	IF Execute
	THEN
		Error												:=	FALSE;
		ErrorId												:= 0;
		CfgReconfigGroup.bExecute 							:= TRUE;
	ELSIF NOT CfgReconfigGroup.bBusy    					
	THEN                                					
		Error												:=	FALSE;
		ErrorId												:= 0;
		CfgReconfigGroup.bExecute 							:= FALSE;

	END_IF

	CfgReconfigGroup(
		bExecute	:= ,
		nGroupId	:= rNCIRef.NciToPlc.GrpId,
		tTimeOut	:= ,
		bBusy		=> busy,
		bErr		=> ,
		nErrId		=> );

	Done													:= NOT CfgReconfigGroup.bBusy
																AND NOT CfgReconfigGroup.bErr
																AND CfgReconfigGroup.bExecute;
                                        					
	IF NOT Busy
	THEN
		IF CfgReconfigGroup.bExecute
		THEN
			Error											:=	CfgReconfigGroup.bErr;
			ErrorId											:= CfgReconfigGroup.nErrId;
			ErrorText										:= SEL(Error , '' ,  CONCAT('Error CfgReconfigGroup id: ',  UDINT_TO_STRING(Errorid)));
		END_IF                      						
		IF NOT Execute              						
		THEN                        						
			MemFnc											:= -1 ;
			CfgReconfigGroup(bExecute := FALSE,);
		END_IF
	END_IF
	
	Reconfig												:= Busy;
END_METHOD

METHOD PUBLIC reconfigAxis : BOOL //Return value = TRUE if busy
//required parameter
//rNCIRef
//AxisId
VAR_INPUT
	Execute													:	BOOL;
	AxisId													:	UDINT; //Axis ID which should be released from group - if 0 then ID of input parameters is used based on parameter AxisIndex
END_VAR
	MemFnc													:= FNC_ADD_AXIS;
	THIS^.Execute											:= Execute;
	
IF NOT __ISVALIDREF(rNCIRef) THEN
	Busy													:= NOT Error;
	Error													:= TRUE;
	ErrorId													:= E_AdsErr.DEVICE_INVALIDPARM;
	Done													:= FALSE;
	ErrorText												:= 'Reference to rNCIRef invalid (0)';
	MemFnc													:= SEL(Execute , -1 ,MemFnc);
	RETURN;
END_IF

	IF Execute
	THEN
		Error												:=	FALSE;
		ErrorId												:= 0;
		CfgReconfigAxis.bExecute 							:= TRUE;
	ELSIF NOT CfgReconfigAxis.bBusy     					
	THEN                                					
		Error												:=	FALSE;
		ErrorId												:= 0;
		CfgReconfigAxis.bExecute 							:= FALSE;

	END_IF

	IF AxisId > 0
	THEN
		CfgReconfigAxis.nAxisId								:= AxisId;
	ELSE
		CASE AxisIndex OF
		1:	CfgReconfigAxis.nAxisId 						:= XAxisId ;
		2:	CfgReconfigAxis.nAxisId 						:= YAxisId ;
		3:	CfgReconfigAxis.nAxisId 						:= ZAxisId ;
		4:	CfgReconfigAxis.nAxisId 						:= Q1AxisId ;
		5:	CfgReconfigAxis.nAxisId 						:= Q2AxisId ;
		6:	CfgReconfigAxis.nAxisId 						:= Q3AxisId ;
		7:	CfgReconfigAxis.nAxisId 						:= Q4AxisId ;
		8:	CfgReconfigAxis.nAxisId 						:= Q5AxisId ;
		ELSE
			CfgReconfigAxis.nAxisId 						:= 0;
		END_CASE
	END_IF

	CfgReconfigAxis(
		bExecute	:= ,
		nAxisId		:= ,
		tTimeOut	:= ,
		bBusy		=> busy,
		bErr		=> ,
		nErrId		=> );

	Done													:= NOT CfgReconfigAxis.bBusy
																AND NOT CfgReconfigAxis.bErr
																AND CfgReconfigAxis.bExecute;
                                        					
	IF NOT Busy
	THEN
		IF CfgReconfigAxis.bExecute
		THEN
			Error											:=	CfgReconfigAxis.bErr;
			ErrorId											:= CfgReconfigAxis.nErrId;
			ErrorText										:= SEL(Error , '' ,  CONCAT('Error CfgReconfigAxis id: ',  UDINT_TO_STRING(Errorid)));
		END_IF
		IF NOT Execute
		THEN
			MemFnc											:= -1 ;
			CfgReconfigAxis(bExecute := FALSE);
		END_IF
	END_IF
	
	ReconfigAxis											:= Busy;
END_METHOD

END_FUNCTION_BLOCK

// POUs/Motion/TF5100-NCI/01_Main/NciItp
//Nci Interpolation group control - load,start,stop Nci programs as well start interpolated moves via Plc table (Tc2_PlcInterpolation library)
//based on Tc2_NCI, TcNcCfg.lib, Tc2_PlcInterpolation librarys
FUNCTION_BLOCK NciItp  EXTENDS FbBase
VAR_OUTPUT CONSTANT
	FNC_RESET												:	INT := 0; //Reset Nci group
	FNC_LOAD												:	INT := 1; //Load Nci program as txt/nc file
	FNC_START												:	INT := 2; //Start loaded Nci program
	FNC_STOP												:	INT := 3; //Stop loaded Nci programm
	FNC_FEED_TBL											:	INT := 4; //Feed table group - provided by Tc2_PlcInterpolation library
END_VAR                     								
VAR_INPUT                   								
	Fnc														:	INT (FNC_RESET..FNC_FEED_TBL):= FNC_RESET;
	Prg														:	T_MaxString := '';	//Program
	rTable													:	REFERENCE TO ST_NciFeedGroupTable := 0; //-> NciItpTableEntry
	rNCIRef													:	REFERENCE TO NCI_REF := 0;
	StartPrgAfterLoading									:	BOOL := FALSE; //Return value TRUE = Start Program direct after loading 
	LogFeederEntries										:	BOOL := FALSE; //Return value TRUE = Log tabel entries by Fnc FeedTbl
	WaitForChnDoneByEndOfTbl								:	BOOL := FALSE; //Fnc FeedTabl - TRUE = FB is busy as long as the prg is running if table contains entry "ST_NciEndOfTables"
END_VAR                     								
VAR_IN_OUT                  								
END_VAR                     								
VAR_OUTPUT                  								
	ErrorText												:	STRING(40);
END_VAR
VAR
(* cache **************************************************************************)
	MemFnc													:	INT := -1;
	MemResetAfterStop										:	BOOL;
                            								
(* timer *)                 								
                            	
(* trigger *)               	

(* MC-Function-block intances ******************************************************)
	ItpLoadProgEx											:	ItpLoadProgEx;
	ItpStartStopEx											:	ItpStartStopEx;
	NciFeedTable											:	FB_NciFeedTable;
	ItpResetEx2												:	ItpResetEx2 := (tTimeOut	:= DEFAULT_ADS_TIMEOUT);

END_VAR

	(* NCI Program control																*)
	(************************************************************************************)

(* Execute ***************************************************************************************)
	rtExecute(CLK := Execute );
	IF rtExecute.Q
		AND MemFnc < 0
	THEN
		MemFnc 												:= Fnc;
		Busy												:= TRUE;
		Done												:= FALSE;
		Error												:= FALSE;
		ErrorID												:= 0;
		ErrorText											:= '';
	END_IF

(* Call Method ***********************************************************************************)
	CASE MemFnc OF
	FNC_RESET							:
		Reset(Execute:= Execute);
	FNC_LOAD							:
		LoadPrg(Execute:= Execute, Prg:= Prg);
	FNC_START							:
		StartPrg(Execute:= Execute);
	FNC_STOP							:
		StopPrg(Execute:= Execute);
	FNC_FEED_TBL						:
		FeedTbl(Execute:= Execute );
	-1:
		IF NOT Execute
		THEN
			Busy											:= FALSE;
			Done											:= FALSE;
			Error											:= FALSE;
			ErrorID											:= 0;
			ErrorText										:= '';
		END_IF                              				
	ELSE                                    				
		Busy												:= FALSE;
		Done												:= FALSE;
		Error												:= Execute;
		ErrorID												:= E_AdsErr.DEVICE_INVALIDPARM;
		ErrorText											:= CONCAT('invalid parameter value(s) Fnc no: ' , INT_TO_STRING(MemFnc));
	END_CASE


(**************************************************************************************************)

METHOD PUBLIC feedTbl : BOOL //Return value = TRUE if busy
//required parameter
//rNCIRef
//rTable
VAR_INPUT
	Execute													:	BOOL := FALSE;
END_VAR
	MemFnc													:= FNC_FEED_TBL;
	THIS^.Execute											:= Execute;
	
IF NOT __ISVALIDREF(rNCIRef) 
THEN
	Busy													:= NOT Error;
	Error													:= TRUE;
	ErrorId													:= E_AdsErr.DEVICE_INVALIDPARM;
	Done													:= FALSE;
	ErrorText												:= 'Reference rNCIRef invalid (0)';
	MemFnc													:= SEL(Execute , -1 ,MemFnc); 
	RETURN;
ELSIF NOT __ISVALIDREF(rTable) 
THEN
	Busy													:= NOT Error;
	Error													:= TRUE;
	ErrorId													:= E_AdsErr.DEVICE_INVALIDPARM;
	Done													:= FALSE;
	ErrorText												:= 'Reference rTable invalid (0)';
	MemFnc													:= SEL(Execute , -1 ,MemFnc);
	RETURN;
END_IF

	IF Execute
	THEN
		Error												:=	FALSE;
		ErrorId												:= 0;
		NciFeedTable.bExecute 								:= TRUE;
	ELSIF NOT NciFeedTable.bFeedBusy
		AND(
		NOT NciFeedTable.bExecChannelDoneCheck
		OR NciFeedTable.bChannelDone)
	THEN
		Error												:=	FALSE;
		ErrorId												:= 0;
		NciFeedTable.bExecute 								:= FALSE;
	END_IF

	NciFeedTable(
		bExecute			:= ,
		bReset				:= FALSE,
		bLogFeederEntries	:= LogFeederEntries,
		stFeedGroupTable	:= rTable,
		stNciToPlc			:= rNCIRef.NciToPlc,
		bFeedingDone		=> 	,
		bChannelDone		=> ,
		bFeedBusy			=> ,
		bResetBusy			=> ,
		bError				=> ,
		nErrorId			=> );

	IF WaitForChnDoneByEndOfTbl
	THEN
		Busy 												:= NciFeedTable.bFeedBusy
																OR
																NciFeedTable.bFeedingDone
																AND NciFeedTable.bExecChannelDoneCheck
																AND NOT NciFeedTable.bChannelDone;
                            								
		Done												:= NciFeedTable.bChannelDone
																OR
																NciFeedTable.bFeedingDone
																AND NOT NciFeedTable.bExecChannelDoneCheck;
                            								
	ELSE                    								
		Busy												:= NciFeedTable.bFeedBusy;
		Done												:= NciFeedTable.bFeedingDone;
	END_IF

	IF NOT Busy
	THEN
		IF NciFeedTable.bExecute
		THEN
			Error											:=	NciFeedTable.bError;
			ErrorId											:= NciFeedTable.nErrorId;
			ErrorText										:= SEL(Error , '' ,  CONCAT('Error NciFeedTable id: ',  UDINT_TO_STRING(Errorid)));
		END_IF                          					
		IF NOT Execute                  					
		THEN                            					
			MemFnc											:= -1 ;
			NciFeedTable(bExecute 							:= FALSE, stNciToPlc:= rNCIRef.NciToPlc, stFeedGroupTable:= rTable  );
		END_IF                          	
	END_IF                              	
                                        	
	FeedTbl													:= Busy;
END_METHOD

METHOD PUBLIC loadPrg : BOOL //Return value = TRUE if busy
//required parameter
//rNCIRef
VAR_INPUT
	Execute													:	BOOL;
	Prg														:	T_MaxString := ''; //if Prg = '' then INPUT THIS^.Prg used
END_VAR
	MemFnc													:= FNC_LOAD;
	THIS^.Execute											:= Execute;
	
IF NOT __ISVALIDREF(rNCIRef) THEN
	Busy													:= NOT Error;
	Error													:= TRUE;
	ErrorId													:= E_AdsErr.DEVICE_INVALIDPARM;
	Done													:= FALSE;
	ErrorText												:= 'Reference rNCIRef invalid (0)';
	MemFnc													:= SEL(Execute , -1 ,MemFnc);
	RETURN;
END_IF
	
	IF Execute AND NOT ItpLoadProgEx.bExecute
	THEN
		IF LEN(Prg) > 0
		THEN
			ItpLoadProgEx.sPrg								:= Prg;
		ELSE                    							
			ItpLoadProgEx.sPrg								:= THIS^.Prg;	
		END_IF
	END_IF	
	
	IF Execute
	THEN
		Error												:=	FALSE;
		ErrorId												:= 0;
		ItpLoadProgEx.bExecute 								:= TRUE;
	ELSIF NOT ItpLoadProgEx.bBusy       					
		AND(                            					
		NOT ItpStartStopEx.bBusy        					
		OR NOT StartPrgAfterLoading)    					
	THEN                                					
		Error												:=	FALSE;
		ErrorId												:= 0;
		ItpLoadProgEx.bExecute 								:= FALSE;
		IF StartPrgAfterLoading             				
		THEN                                				
			ItpStartStopEx.bStart 							:= FALSE;
		END_IF
	END_IF
	
	ItpLoadProgEx(
		bExecute	:= ,
		sPrg		:= ,
		nLength		:= INT_TO_UDINT(LEN(Prg)),
		tTimeOut	:= ,
		sNciToPlc	:= rNCIRef.NciToPlc,
		bBusy		=> ,
		bErr		=> ,
		nErrId		=> );

	IF StartPrgAfterLoading
		OR ItpStartStopEx.bBusy
	THEN
		ItpStartStopEx(
			bStart		:= ItpLoadProgEx.bExecute
							AND NOT ItpLoadProgEx.bErr
							AND NOT ItpLoadProgEx.bBusy,
			bStop		:= FALSE,
			tTimeOut	:=  ,
			sNciToPlc	:= rNCIRef.NciToPlc,
			bBusy		=> ,
			bErr		=> ,
			nErrId		=> );
	END_IF


	Busy													:= ItpStartStopEx.bBusy OR ItpLoadProgEx.bBusy;
                                        					
	IF StartPrgAfterLoading             					
	THEN                                					
		Done												:= NOT Busy
																AND NOT ItpStartStopEx.bErr
																AND ItpStartStopEx.bStart;
	ELSE                                	    		
		Done												:= NOT Busy
																AND NOT ItpLoadProgEx.bErr
																AND ItpLoadProgEx.bExecute;
	END_IF                                      		
                                                	
	IF NOT Busy                                 	
	THEN
		IF ItpLoadProgEx.bExecute
			AND NOT StartPrgAfterLoading
		THEN
			Error											:=	ItpLoadProgEx.bErr;
			ErrorId											:= ItpLoadProgEx.nErrId;
			ErrorText										:= SEL(Error , '' ,  CONCAT('Error ItpLoadProgEx id: ',  UDINT_TO_STRING(Errorid)));
		ELSIF ItpStartStopEx.bStart 						
		THEN                        						
			Error												:=	ItpStartStopEx.bErr;
			ErrorId											:= ItpStartStopEx.nErrId;
			ErrorText										:= SEL(Error , '' ,  CONCAT('Error ItpStartStopEx id: ',  UDINT_TO_STRING(Errorid)));
		END_IF                          					
                                        					
		IF NOT Execute                  	
		THEN                            	
			MemFnc											:= -1 ;
			ItpLoadProgEx(bExecute := FALSE, sNciToPlc:= rNCIRef.NciToPlc);
			IF StartPrgAfterLoading
			THEN
				ItpStartStopEx(bStart := FALSE, sNciToPlc:= rNCIRef.NciToPlc);
			END_IF
		END_IF
	END_IF
	
	LoadPrg													:= Busy;
END_METHOD

METHOD PUBLIC reset : BOOL //Return value = TRUE if busy
//required parameter
//rNCIRef
//rTable
VAR_INPUT	
	Execute													:	BOOL := FALSE;
END_VAR
	MemFnc													:= FNC_RESET;
	THIS^.Execute											:= Execute;
	
IF NOT __ISVALIDREF(rNCIRef) 
THEN
	Busy													:= NOT Error;
	Error													:= TRUE;
	ErrorId													:= E_AdsErr.DEVICE_INVALIDPARM;
	Done													:= FALSE;
	ErrorText												:= 'Reference rNCIRef invalid (0)';
	MemFnc													:= SEL(Execute , -1 ,MemFnc);
	RETURN;
ELSIF NOT __ISVALIDREF(rTable) AND FALSE 
THEN
	Busy													:= NOT Error;
	Error													:= TRUE;
	ErrorId													:= E_AdsErr.DEVICE_INVALIDPARM;
	Done													:= FALSE;
	ErrorText												:= 'Reference rTable invalid (0)';
	MemFnc													:= SEL(Execute , -1 ,MemFnc);
	RETURN;
END_IF

IF Execute
THEN
	Error													:=	FALSE;
	ErrorId													:= 0;
	NciFeedTable.bReset 									:= __ISVALIDREF(rTable);
	ItpResetEx2.bExecute									:= NOT __ISVALIDREF(rTable);
ELSIF NOT NciFeedTable.bFeedBusy                        	
AND NOT ItpResetEx2.bBusy                               	
THEN                                                    	
	Error													:=	FALSE;
	ErrorId													:= 0;
	NciFeedTable.bReset 									:= FALSE;
	ItpResetEx2.bExecute									:= FALSE; 
END_IF

IF	NOT __ISVALIDREF(rTable)
THEN
	ItpResetEx2(
		bExecute	:= ,
		tTimeOut	:= ,
		sNciToPlc	:= rNCIRef.NciToPlc,
		bBusy		=> Busy,
		bErr		=> ,
		nErrId		=> );
ELSE
	NciFeedTable(
		bExecute			:= FALSE,
		bReset				:= ,
		bLogFeederEntries	:= ,
		stFeedGroupTable	:= rTable,
		stNciToPlc			:= rNCIRef.NciToPlc,
		bFeedingDone		=> ,
		bChannelDone		=> ,
		bFeedBusy			=> ,
		bResetBusy			=> busy,
		bError				=> ,
		nErrorId			=> );
END_IF
Done														:= NOT NciFeedTable.bResetBusy AND NOT ItpResetEx2.bBusy
															 	AND NOT NciFeedTable.bError AND NOT ItpResetEx2.bErr
															 	AND(NciFeedTable.bReset OR ItpResetEx2.bExecute);
                                                      	     
IF NOT Busy                                           	     
THEN                                                  	     
	IF NciFeedTable.bReset                            	     
	THEN                                              	     
		Error												 :=	NciFeedTable.bError;
		ErrorId												 := NciFeedTable.nErrorId;
		ErrorText											 := SEL(Error , '' ,  CONCAT('Error NciFeedTable id: ',  UDINT_TO_STRING(Errorid)));
	ELSIF ItpResetEx2.bExecute      						 
	THEN                            						 
		Error												 :=	ItpResetEx2.bErr;
		ErrorId												 := ItpResetEx2.nErrId;
		ErrorText											 := SEL(Error , '' ,  CONCAT('Error ItpResetEx2 id: ',  UDINT_TO_STRING(Errorid)));		
	END_IF                                            	     
	IF NOT Execute                                    	     
	THEN                                                	
		MemFnc												:= -1 ;
		IF	NOT __ISVALIDREF(rTable)                    	
		THEN                                            	
			ItpResetEx2(bExecute							:= FALSE,sNciToPlc:= rNCIRef.NciToPlc);
		ELSE                                            	
			NciFeedTable(bReset 							:= FALSE, stNciToPlc:= rNCIRef.NciToPlc,stFeedGroupTable:= rTable );
		END_IF                                          	
	END_IF                                              	
END_IF                                                  	
                                                        	
Reset														:= Busy;
END_METHOD

METHOD PUBLIC startPrg : BOOL //Return value = TRUE if busy
//required parameter
//rNCIRef
VAR_INPUT
	Execute													:	BOOL;
END_VAR
	MemFnc													:= FNC_START;
	THIS^.Execute											:= Execute;
	
IF NOT __ISVALIDREF(rNCIRef) THEN
	Busy													:= NOT Error;
	Error													:= TRUE;
	ErrorId													:= E_AdsErr.DEVICE_INVALIDPARM;
	Done													:= FALSE;
	ErrorText												:= 'Reference rNCIRef invalid (0)';
	MemFnc													:= SEL(Execute , -1 ,MemFnc);
	RETURN;
END_IF

	IF Execute
	THEN
		Error												:=	FALSE;
		ErrorId												:= 0;
		ItpStartStopEx.bStart 								:= TRUE;
	ELSIF NOT ItpStartStopEx.bBusy      					
	THEN                                					
		Error												:=	FALSE;
		ErrorId												:= 0;
		ItpStartStopEx.bStart 								:= FALSE;

	END_IF
	
	ItpStartStopEx(
		bStart		:= ,
		bStop		:= FALSE,
		tTimeOut	:=  ,
		sNciToPlc:= rNCIRef.NciToPlc,
		bBusy		=> busy,
		bErr		=> ,
		nErrId		=> );


	Done													:= NOT ItpStartStopEx.bBusy
																AND NOT ItpStartStopEx.bErr
																AND ItpStartStopEx.bStart;
                                        					
	IF NOT Busy
	THEN
		IF ItpStartStopEx.bStart
		THEN
			Error											:=	ItpStartStopEx.bErr;
			ErrorId											:= ItpStartStopEx.nErrId;
			ErrorText										:= SEL(Error , '' ,  CONCAT('Error ItpStartStopEx id: ',  UDINT_TO_STRING(Errorid)));
		END_IF
		IF NOT Execute
		THEN
			MemFnc											:= -1 ;
			ItpStartStopEx(bStart := FALSE, sNciToPlc:= rNCIRef.NciToPlc);
		END_IF
	END_IF
	
	StartPrg												:= Busy;
END_METHOD

METHOD PUBLIC stopPrg : BOOL //Return value = TRUE if busy
//required parameter
//rNCIRef
//rTable
VAR_INPUT
	Execute													:	BOOL;
END_VAR
	MemFnc													:= FNC_STOP;
	THIS^.Execute											:= Execute;
	
IF NOT __ISVALIDREF(rNCIRef) THEN
	Busy													:= NOT Error;
	Error													:= TRUE;
	ErrorId													:= E_AdsErr.DEVICE_INVALIDPARM;
	Done													:= FALSE;
	ErrorText												:= 'Reference rNCIRef invalid (0)';
	MemFnc													:= SEL(Execute , -1 ,MemFnc);
	RETURN;
END_IF

	IF Execute
	THEN
		Error												:=	FALSE;
		ErrorId												:= 0;
		ItpStartStopEx.bStop 								:= TRUE;
	ELSIF NOT ItpStartStopEx.bBusy      					
		AND NOT NciFeedTable.bResetBusy 					
	THEN                                					
		Error												:=	FALSE;
		ErrorId												:= 0;
		ItpStartStopEx.bStop 								:= FALSE;
	END_IF

	ItpStartStopEx(
		bStart		:= FALSE,
		bStop		:= ,
		tTimeOut	:=  ,
		sNciToPlc	:= rNCIRef.NciToPlc,
		bBusy		=> ,
		bErr		=> ,
		nErrId		=> );

	IF ItpStartStopEx.bStop
		AND ItpStartStopEx.bBusy
		AND rNCIRef.NciToPlc.ItpState > NCI_INTERPRETER_READY
		AND rNCIRef.NciToPlc.ItpState <> NCI_INTERPRETER_ABORTED
	THEN (* After stopping an active programm, please reset the function-block to avoid the error 0x42C5 after restart *)
		MemResetAfterStop 									:= TRUE;
	END_IF

	NciFeedTable(
		bExecute		:= FALSE,
		bReset			:= NOT ItpStartStopEx.bBusy
								AND NOT ItpStartStopEx.bErr
								AND ItpStartStopEx.bStop
								AND MemResetAfterStop,
		bLogFeederEntries:= ,
		stFeedGroupTable:= rTable,
		stNciToPlc		:= rNCIRef.NciToPlc,
		bFeedingDone	=> ,
		bChannelDone	=> ,
		bFeedBusy		=> ,
		bResetBusy		=> ,
		bError			=> ,
		nErrorId			=> );

	Busy													:= NciFeedTable.bResetBusy OR ItpStartStopEx.bBusy;
                                        					
	Done													:= NOT Busy
																AND NOT ItpStartStopEx.bErr
																AND ItpStartStopEx.bStop;

	IF NOT Busy
	THEN
		IF ItpStartStopEx.bStop
		THEN
			Error											:=	ItpStartStopEx.bErr;
			ErrorId											:= ItpStartStopEx.nErrId;
			ErrorText										:= SEL(Error , '' ,  CONCAT('Error ItpStartStopEx id: ',  UDINT_TO_STRING(Errorid)));
		END_IF
		IF NOT Execute
		THEN
			MemResetAfterStop								:= FALSE;
			MemFnc											:= -1 ;
			ItpStartStopEx(bStop 							:= FALSE, sNciToPlc:= rNCIRef.NciToPlc);
			NciFeedTable(bExecute 							:= FALSE, stNciToPlc:= rNCIRef.NciToPlc,stFeedGroupTable:= rTable );
		END_IF                      						
	END_IF                          						
	                                	
	StopPrg													:= Busy;
END_METHOD

END_FUNCTION_BLOCK

// POUs/Motion/TF5100-NCI/01_Main/NciMotion
{attribute 'no_check'}
//Nci group motion control - Send EStop to group, release EStop via StepOn command, backup Nci program to make use of start retrace program forward/backward  
//based on Tc2_NCI
FUNCTION_BLOCK NciMotion  EXTENDS FbBase
VAR_OUTPUT CONSTANT
	FNC_ESTOP												:	INT := 0; //Send EStop to Nci group 
	FNC_STEP_ON												:	INT := 1; 
	FNC_ENABLE_FEEDER_BACKUP								:	INT := 2;
	FNC_DISABLE_FEEDER_BACKUP								:	INT := 3;
	FNC_RETRACE_FWD											:	INT := 4;
	FNC_RETRACE_BWD											:	INT := 5;
END_VAR                         							
VAR_INPUT                       							
	Fnc														:	INT (FNC_ESTOP..FNC_RETRACE_BWD):= FNC_ESTOP;
	rNCIRef													:	REFERENCE TO NCI_REF := 0;
END_VAR
VAR_IN_OUT
END_VAR
VAR_OUTPUT
	ErrorText												:	STRING(40);	
END_VAR
VAR
(* cache **************************************************************************)
	MemFnc													:	INT := -1;

(* Timer *)


(* Trigger *)

(* MC-functionblock instances *******************************************************)
	ItpRetraceMoveBackward									:	ItpRetraceMoveBackward := (tTimeOut	:= DEFAULT_ADS_TIMEOUT);
	ItpRetraceMoveForward									: 	ItpRetraceMoveForward := (tTimeOut	:= DEFAULT_ADS_TIMEOUT);
	ItpEStopEx												:	ItpEStopEx := (tTimeOut	:= DEFAULT_ADS_TIMEOUT);
	ItpStepOnAfterEStopEx									:	ItpStepOnAfterEStopEx := (tTimeOut	:= DEFAULT_ADS_TIMEOUT);
	ItpEnableFeederBackup									:	ItpEnableFeederBackup := (tTimeOut	:= DEFAULT_ADS_TIMEOUT);

END_VAR

	(* Nci group control																*)
	(************************************************************************************)

(* Execute ***************************************************************************************)
	rtExecute(CLK := Execute );
	IF rtExecute.Q
		AND MemFnc < 0
	THEN
		MemFnc 												:= Fnc;
		Busy												:= TRUE;
		Done												:= FALSE;
		Error												:= FALSE;
		ErrorID												:= 0;
		ErrorText											:= '';
	END_IF

(* Call Method ***********************************************************************************)
	CASE MemFnc OF
	FNC_ESTOP												:	EStop(Execute);
	FNC_STEP_ON												:	StepOn(Execute);
	FNC_ENABLE_FEEDER_BACKUP								:	EnableFeederBackup(Execute);
	FNC_DISABLE_FEEDER_BACKUP								:	DisableFeederBackup(Execute);
	FNC_RETRACE_FWD											:	RetraceFwd(Execute);
	FNC_RETRACE_BWD											:	RetraceBwd(Execute);
	-1:
		IF NOT Execute
		THEN
			Busy											:= FALSE;
			Done											:= FALSE;
			Error											:= FALSE;
			ErrorID											:= 0;
			ErrorText										:= '';
		END_IF                              				
	ELSE                                    				
		Busy												:= FALSE;
		Done												:= FALSE;
		Error												:= Execute;
		ErrorID												:= E_AdsErr.DEVICE_INVALIDPARM;
		ErrorText											:= CONCAT('invalid parameter value(s) Fnc no: ' , INT_TO_STRING(MemFnc));
	END_CASE

(**************************************************************************************************)

METHOD PUBLIC disableFeederBackup : BOOL //Return value = TRUE if busy
//required parameter
//rNCIRef
VAR_INPUT
	Execute													:	BOOL;
END_VAR
	MemFnc													:= FNC_DISABLE_FEEDER_BACKUP;
	THIS^.Execute											:= Execute;
	                                                    	
IF NOT __ISVALIDREF(rNCIRef)                            	
THEN                                                    	
	Busy													:= NOT Error;
	Error													:= TRUE;
	ErrorId													:= E_AdsErr.DEVICE_INVALIDPARM;
	Done													:= FALSE;
	ErrorText												:= 'Reference to rNCIRef invalid (0)';
	MemFnc													:= SEL(Execute , -1 ,MemFnc); 
	RETURN;
END_IF

IF Execute
THEN
	Error													:=	FALSE;
	ErrorId													:= 0;
	ItpEnableFeederBackup.bExecute 							:= TRUE;
ELSIF NOT ItpEnableFeederBackup.bBusy   					
THEN                                    					
	Error													:=	FALSE;
	ErrorId													:= 0;
	ItpEnableFeederBackup.bExecute 							:= FALSE;
                                                        	
END_IF                                                  	
                                                        	
ItpEnableFeederBackup(                                  	
	bEnable		:= FALSE,                               	
	bExecute	:= ,                                    	
	tTimeOut	:= ,                                    	
	sNciToPlc	:= rNCIRef.NciToPlc,                    	
	bBusy		=> busy,                                	
	bErr		=> ,                                    	
	nErrId		=> );                                   	
                                                        	
Done														:= NOT ItpEnableFeederBackup.bBusy
																AND NOT ItpEnableFeederBackup.bErr
																AND ItpEnableFeederBackup.bExecute;
                                                        	
IF NOT Busy                                             	
THEN                                                    	
	IF ItpEnableFeederBackup.bExecute                   	
	THEN                                                	
		Error												:=	ItpEnableFeederBackup.bErr;
		ErrorId												:= ItpEnableFeederBackup.nErrId;
		ErrorText											:= SEL(Error , '' ,  CONCAT('Error ItpEnableFeederBackup (EN=FALSE) id: ',  UDINT_TO_STRING(Errorid)));
	END_IF                          						
	IF NOT Execute                  						
	THEN                            	                		
		MemFnc												:= -1 ;
		ItpEnableFeederBackup(bExecute := FALSE, sNciToPlc:= rNCIRef.NciToPlc);
	END_IF
END_IF

DisableFeederBackup											:= FALSE;
END_METHOD

METHOD PUBLIC enableFeederBackup : BOOL //Return value = TRUE if busy
//required parameter
//rNCIRef
VAR_INPUT
	Execute													:	BOOL;
END_VAR
	MemFnc													:= FNC_DISABLE_FEEDER_BACKUP;
	THIS^.Execute											:= Execute;
	
IF NOT __ISVALIDREF(rNCIRef) 
THEN
	Busy													:= NOT Error;
	Error													:= TRUE;
	ErrorId													:= E_AdsErr.DEVICE_INVALIDPARM;
	Done													:= FALSE;
	ErrorText												:= 'Reference to rNCIRef invalid (0)';
	MemFnc													:= SEL(Execute , -1 ,MemFnc); 
	RETURN;
END_IF

	IF Execute
	THEN
		Error												:=	FALSE;
		ErrorId												:= 0;
		ItpEnableFeederBackup.bExecute 						:= TRUE;
	ELSIF NOT ItpEnableFeederBackup.bBusy   				
	THEN                                    				
		Error												:=	FALSE;
		ErrorId												:= 0;
		ItpEnableFeederBackup.bExecute 						:= FALSE;

	END_IF

	ItpEnableFeederBackup(
		bEnable		:= TRUE,
		bExecute	:= ,
		tTimeOut	:= ,
		sNciToPlc	:= rNCIRef.NciToPlc,
		bBusy		=> busy,
		bErr		=> ,
		nErrId		=> );

	Done													:= NOT ItpEnableFeederBackup.bBusy
																AND NOT ItpEnableFeederBackup.bErr
																AND ItpEnableFeederBackup.bExecute;

	IF NOT Busy
	THEN
		IF ItpEnableFeederBackup.bExecute
		THEN
			Error											:=	ItpEnableFeederBackup.bErr;
			ErrorId											:= ItpEnableFeederBackup.nErrId;
			ErrorText										:= SEL(Error , '' ,  CONCAT('Error ItpEnableFeederBackup (EN=TRUE) id: ',  UDINT_TO_STRING(Errorid)));
		END_IF
		IF NOT Execute
		THEN
			MemFnc											:= -1 ;
			ItpEnableFeederBackup(bExecute := FALSE , sNciToPlc:= rNCIRef.NciToPlc);
		END_IF
	END_IF
	
	EnableFeederBackup										:= Busy;
END_METHOD

METHOD PUBLIC eStop : BOOL //Return value = TRUE if busy
//required parameter
//rNCIRef
VAR_INPUT
	Execute													:	BOOL;
END_VAR
	MemFnc													:= FNC_ESTOP;
	THIS^.Execute											:= Execute;
	
IF NOT __ISVALIDREF(rNCIRef) 
THEN
	Busy													:= NOT Error;
	Error													:= TRUE;
	ErrorId													:= E_AdsErr.DEVICE_INVALIDPARM;
	Done													:= FALSE;
	ErrorText												:= 'Reference to rNCIRef invalid (0)';
	MemFnc													:= -1 ;
	RETURN;
END_IF

	IF Execute
	THEN
		Error												:=	FALSE;
		ErrorId												:= 0;
		ItpEStopEx.bExecute 								:= TRUE;
	ELSIF NOT ItpEStopEx.bBusy          					
	THEN                                					
		Error												:=	FALSE;
		ErrorId												:= 0;
		ItpEStopEx.bExecute 								:= FALSE;

	END_IF
	
	ItpEStopEx(
		bExecute	:= ,
		fDec		:= (* Dec *),
		fJerk		:= (* Jerk *),
		tTimeOut	:= ,
		sNciToPlc	:= rNCIRef.NciToPlc,
		bBusy		=> Busy,
		bErr		=> ,
		nErrId	=> );

	Done													:= NOT ItpEStopEx.bBusy
																AND NOT ItpEStopEx.bErr
																AND ItpEStopEx.bExecute;

	IF NOT Busy
	THEN
		IF ItpEStopEx.bExecute
		THEN
			Error											:=	ItpEStopEx.bErr;
			ErrorId											:= ItpEStopEx.nErrId;
			ErrorText										:= SEL(Error , '' ,  CONCAT('Error ItpEStopEx id: ',  UDINT_TO_STRING(Errorid)));
		END_IF
		IF NOT Execute
		THEN
			MemFnc											:= -1 ;
			ItpEStopEx(bExecute := FALSE, sNciToPlc:= rNCIRef.NciToPlc);
		END_IF
	END_IF

	EStop													:= Busy;
END_METHOD

METHOD PUBLIC retraceBwd : BOOL //Return value = TRUE if busy
//required parameter
//rNCIRef
VAR_INPUT
	Execute													:	BOOL;
END_VAR
	MemFnc													:= FNC_RETRACE_BWD;
	THIS^.Execute											:= Execute;
	
IF NOT __ISVALIDREF(rNCIRef) THEN
	Busy													:= NOT Error;
	Error													:= TRUE;
	ErrorId													:= 16#4B30;
	Done													:= FALSE;
	ErrorText												:= 'Reference to rNCIRef invalid (0)';
	MemFnc													:= SEL(Execute , -1 ,MemFnc); 
	RETURN;
END_IF

IF Execute
THEN
	Error												:=	FALSE;
	ErrorId												:= 0;
	ItpRetraceMoveBackward.bExecute 					:= TRUE;
ELSIF NOT ItpRetraceMoveBackward.bBusy      			
THEN                                        			
	Error												:=	FALSE;
	ErrorId												:= 0;
ItpRetraceMoveBackward.bExecute 						:= FALSE;

END_IF

ItpRetraceMoveBackward(
	bExecute	:= ,
	tTimeOut	:= ,
	sNciToPlc	:= rNCIRef.NciToPlc,
	bBusy		=> Busy,
	bErr		=> ,
	nErrId		=> );
Done													:= NOT ItpRetraceMoveBackward.bBusy
															AND NOT ItpRetraceMoveBackward.bErr
															AND ItpRetraceMoveBackward.bExecute;

IF NOT Busy
THEN
	IF ItpRetraceMoveBackward.bExecute
	THEN
		Error											:=	ItpRetraceMoveBackward.bErr;
		ErrorId											:= ItpRetraceMoveBackward.nErrId;
		ErrorText										:= SEL(Error , '' ,  CONCAT('Error ItpRetraceMoveBackward id: ',  UDINT_TO_STRING(Errorid)));
	END_IF
	IF NOT Execute
	THEN
		MemFnc											:= -1 ;
		ItpRetraceMoveBackward(bExecute := FALSE, sNciToPlc:= rNCIRef.NciToPlc);
	END_IF
END_IF

RetraceBwd												:= Busy;
END_METHOD

METHOD PUBLIC retraceFwd : BOOL //Return value = TRUE if busy
//required parameter
//rNCIRef
VAR_INPUT
	Execute													:	BOOL;
END_VAR
	MemFnc													:= FNC_RETRACE_FWD;
	THIS^.Execute											:= Execute;
IF NOT __ISVALIDREF(rNCIRef) 
THEN
	Busy													:= NOT Error;
	Error													:= TRUE;
	ErrorId													:= E_AdsErr.DEVICE_INVALIDPARM;
	Done													:= FALSE;
	ErrorText												:= 'Reference to rNCIRef invalid (0)';
	MemFnc													:= SEL(Execute , -1 ,MemFnc); 
	RETURN;
END_IF

	IF Execute
	THEN
		Error												:=	FALSE;
		ErrorId												:= 0;
		ItpRetraceMoveForward.bExecute 						:= TRUE;
	ELSIF NOT ItpRetraceMoveForward.bBusy       			
	THEN                                        			
		Error												:=	FALSE;
		ErrorId												:= 0;
		ItpRetraceMoveForward.bExecute 						:= FALSE;

	END_IF
	
	ItpRetraceMoveForward(
		bExecute	:= ,
		tTimeOut	:= ,
		sNciToPlc	:= rNCIRef.NciToPlc,
		bBusy		=> Busy,
		bErr		=> ,
		nErrId		=> );

	Done												:= NOT ItpRetraceMoveForward.bBusy
															AND NOT ItpRetraceMoveForward.bErr
															AND ItpRetraceMoveForward.bExecute;
                                        				
	IF NOT Busy
	THEN
		IF ItpRetraceMoveForward.bExecute
		THEN
			Error										:=	ItpRetraceMoveForward.bErr;
			ErrorId										:= ItpRetraceMoveForward.nErrId;
			ErrorText									:= SEL(Error , '' ,  CONCAT('Error ItpRetraceMoveForward id: ',  UDINT_TO_STRING(Errorid)));
		END_IF                          				
		IF NOT Execute                  				
		THEN                            	
			MemFnc										:= -1 ;
			ItpRetraceMoveForward(bExecute := FALSE, sNciToPlc:= rNCIRef.NciToPlc);
		END_IF
	END_IF

	RetraceFwd											:= Busy;
END_METHOD

METHOD PUBLIC stepOn : BOOL //Return value = TRUE if busy
//required parameter
//rNCIRef
VAR_INPUT
	Execute													:	BOOL;
END_VAR
	MemFnc													:= FNC_STEP_ON;
	THIS^.Execute											:= Execute;
	
IF NOT __ISVALIDREF(rNCIRef) THEN
	Busy													:= NOT Error;
	Error													:= TRUE;
	ErrorId													:= E_AdsErr.DEVICE_INVALIDPARM;
	Done													:= FALSE;
	ErrorText												:= 'Reference to rNCIRef invalid (0)';
	MemFnc													:= SEL(Execute , -1 ,MemFnc); 
	RETURN;
END_IF

	IF Execute
	THEN
		Error												:=	FALSE;
		ErrorId												:= 0;
		ItpStepOnAfterEStopEx.bExecute 						:= TRUE;
	ELSIF NOT ItpStepOnAfterEStopEx.bBusy   				
	THEN                                    				
		Error												:=	FALSE;
		ErrorId												:= 0;
		ItpStepOnAfterEStopEx.bExecute 						:= FALSE;

	END_IF

	ItpStepOnAfterEStopEx(
		bExecute	:= ,
		tTimeOut	:= ,
		sNciToPlc	:= rNCIRef.NciToPlc,
		bBusy		=> Busy,
		bErr		=> ,
		nErrId		=> );

	Done													:= NOT ItpStepOnAfterEStopEx.bBusy
																AND NOT ItpStepOnAfterEStopEx.bErr
																AND ItpStepOnAfterEStopEx.bExecute;

	IF NOT Busy
	THEN
		IF ItpStepOnAfterEStopEx.bExecute
		THEN
			Error											:=	ItpStepOnAfterEStopEx.bErr;
			ErrorId											:= ItpStepOnAfterEStopEx.nErrId;
			ErrorText										:= SEL(Error , '' ,  CONCAT('Error ItpStepOnAfterEStopEx id: ',  UDINT_TO_STRING(Errorid)));
		END_IF
		IF NOT Execute
		THEN
			MemFnc											:= -1 ;
			ItpStepOnAfterEStopEx(bExecute := FALSE, sNciToPlc:= rNCIRef.NciToPlc);
		END_IF
	END_IF

	stepOn													:= Busy;
END_METHOD

END_FUNCTION_BLOCK

// POUs/Motion/TF5100-NCI/02_Options/Error/NciChnEventHandling
{attribute 'no_check'}
FUNCTION_BLOCK NciChnEventHandling
VAR_INPUT
	Flag													:	BOOL := FALSE;
	ConfirmTrig												:	BOOL;
	MsgId													:	UDINT := 200; //Default
	SourceId												:	UDINT := 101200;
	ChannelId												:	DWORD := 2;
{attribute 'displaymode':='hex'}
	ErrorId													:	UDINT;
	Name													: 	STRING(20);
END_VAR                         							
VAR_OUTPUT                      							
	State													:	UDINT := TCEVENTSTATE_INVALID;
																		(* TCEVENTSTATE_INVALID  	: WORD := 16#0000; (* Ungültig, kommt auch wenn Event noch nicht gemeldet. *)
																			TCEVENTSTATE_SIGNALED  	: WORD := 16#0001; (* Event ist gemeldet, aber weder gegangen noch quittiert. *)
																			TCEVENTSTATE_RESET  		: WORD := 16#0002; (* Event ist abgemeldet ('gegangen'). *)
																			TCEVENTSTATE_CONFIRMED  : WORD := 16#0010 (16); (* Event ist quittiert. *)
																			TCEVENTSTATE_RESETCON  	: WORD := 16#0012 (17); (* Event ist abgemeldet und quittiert *) *)
{attribute 'displaymode':='binary'}
	Status													:	DWORD; (*	.0 - .8 = event <class id>  / .15 Quit required / .16 = Level 0 , .17 = Level 1 , .18 = Level 2, .......... / .31 active
																			TCEVENTCLASS_NONE			:=0,	(* No class *)
																			TCEVENTCLASS_MAINTENANCE	:=1,	(* Maintenance hint *)
																			TCEVENTCLASS_MESSAGE		:=2,	(* Message *)
																			TCEVENTCLASS_HINT			:=3,	(* Hint *)
																			TCEVENTCLASS_STATEINFO		:=4,	(* State information *)
																			TCEVENTCLASS_INSTRUCTION	:=5,	(* Instruction *)
																			TCEVENTCLASS_WARNING		:=6,	(* Warning *)
																			TCEVENTCLASS_ALARM			:=7,	(* Alarm *)
																			TCEVENTCLASS_PARAMERROR		:=8		(* Parameter error *)  *)
END_VAR
VAR
	AdsEvent												:		ADSLOGEVENT :=(
																		Event			:= FALSE,
																		NETID			:= '',
																		PORT			:= AMSPORT_EVENTLOG,
																		TMOUT 			:= DEFAULT_ADS_TIMEOUT,
																		EventConfigData := (
																					Class 			:= TC2_SYSTEM.TCEVENTCLASS_ALARM,
																					Prio 			:= TCEVENTPRIO_IMPLICIT,
																					ProgId 			:= 'TcEventFormatter.TcXmlFormatter',
																					Flags 			:= 16#0140 (* TCEVENTFLAG_LOG OR TCEVENTFLAG_SRCID *),
																					StreamType 		:= TCEVENTSTREAM_NORMAL (* TCEVENTSTREAM_SIMPLE *),
																					bQuitRequired 	:= FALSE));
                    										
	FormatString 											: STRING(15) := '%s%d%s%s%d%s';
                    										
	pParaArray												: ARRAY [1..6] OF PVOID;
                    										
	Para1													: STRING(30);
	Para2													: UDINT;
	Para3													: STRING(70);
	Para4													: STRING(70);
	Para5													: UDINT;
	Para6													: STRING(20);
	SetClass												: E_TcEventClass := TC2_SYSTEM.TCEVENTCLASS_ALARM;
END_VAR

(* Send axis error text to EventLogger		 							*)
(************************************************************************)

(* Event Config ************************************************)
	IF Status.31 //Message active
	THEN (* work EventLogger *)

		AdsEvent(
			NETID			:= ,(* siehe deklaration *)
			PORT			:= ,(* siehe deklaration *)
			Event			:= NOT AdsEvent.FbCleanup AND(Flag AND Para2 = ErrorID OR AdsEvent.EventState = TCEVENTSTATE_INVALID AND NOT AdsEvent.Quit),
			EventQuit		:= AdsEvent.EventState <> TCEVENTSTATE_INVALID
								AND AdsEvent.EventConfigData.bQuitRequired
								AND NOT AdsEvent.Eventstate.4
								AND NOT AdsEvent.Quit
								AND(
								ConfirmTrig
								OR Para2 <> ErrorID
								OR AdsEvent.EventQuit), (* quit send *)
			EventConfigData	:= ,(* siehe deklaration *)
			EventDataAddress:= ADR(pParaArray),
			EventDataLength	:= ,
			FbCleanup		:= NOT AdsEvent.FbCleanup AND(AdsEvent.Err OR AdsEvent.EventState = TCEVENTSTATE_RESETCON),
			TMOUT			:= ,(* siehe deklaration *)
			EventState		=> ,
			Err				=> ,
			ErrId			=> ,
			Quit			=> );

		IF AdsEvent.Event
			AND AdsEvent.EventState = TCEVENTSTATE_INVALID
		THEN
			State 											:= SEL(Flag, TCEVENTSTATE_RESET, TCEVENTSTATE_SIGNALED);
		ELSIF AdsEvent.Quit
			AND AdsEvent.EventState = TCEVENTSTATE_INVALID
			AND AdsEvent.EventQuit
			OR 
			AdsEvent.FbCleanup		
		THEN
			State 											:= TCEVENTSTATE_RESETCON;
		ELSIF(AdsEvent.Err OR NOT AdsEvent.Event AND AdsEvent.EventState = TCEVENTSTATE_INVALID)
			AND_THEN Gvl.EventHandlingStatistic.CountOut(Status)
		THEN
			State											:= TCEVENTSTATE_INVALID;
		ELSE
			State											:= MAX(State, AdsEvent.EventState);
		END_IF
	
	ELSIF flag AND SourceId > 0
	THEN (* fire event *)
	(*	Type : 2 - Axis Event 201
		%1 User Name 
		%2 	Unique error id (DINT)
		%3	Error text (STRING) ) Bsp.: [S750E20392]
		@V1:%4	Error description (STRING) Bsp.: [S751E20392]
		%5	Logical axis id (DINT)
		@V2:%6	Position OF axis (REAL) or Reserved text 
	
	*)
		Para1 												:= Name;
		Para2 												:= ErrorID;
              												
		Para3 												:= CONCAT('[S','700'); (* SOURCE_TEXT_PTPNCI = 701 *)
		Para3 												:= CONCAT(Para3,'E');
		Para3 												:= CONCAT(Para3,UDINT_TO_STRING(ErrorID));
		Para3 												:= CONCAT(Para3,']');
              												
		Para4 												:= CONCAT('[S','701'); (* SOURCE_DESC_PTPNCI = 701 *)
		Para4 												:= CONCAT(Para4,'E');
		Para4 												:= CONCAT(Para4,UDINT_TO_STRING(ErrorID));
		Para4 												:= CONCAT(Para4,']');
              												
		Para5 												:= ChannelId;
		Para6 												:= ''; (* Reserve *)

		pParaArray[1] 										:= ADR(Para1);
		pParaArray[2] 										:= ADR(Para2);
		pParaArray[3] 										:= ADR(Para3);
		pParaArray[4] 										:= ADR(Para4);
		pParaArray[5] 										:= ADR(Para5);
		pParaArray[6] 										:= ADR(Para6);

		
		AdsEvent.EventConfigData.Id 						:= MsgId; (* MSG_ID = 201 *)
 		AdsEvent.EventConfigData.DataFormatStrAddress 		:= ADR(FormatString);
		AdsEvent.EventConfigData.SourceId 					:= SourceId + ChannelId;
		Status												:= Gvl.EventHandlingStatistic.InitEvent(SetClass , AdsEvent.EventConfigData);	

		IF AdsEvent.Err AND NOT AdsEvent.FbCleanup
		THEN
			AdsEvent(
				Event			:= FALSE,
				EventQuit 		:= FALSE,
				EventDataAddress:= ADR(pParaArray),
				FbCleanup		:= TRUE,
				EventState		=> );
		
		ELSE (* Fire Event *)
			AdsEvent( 	Event			:= FALSE,
						EventQuit 		:= FALSE, 
						FbCleanup 		:= FALSE, 
						EventDataAddress:= ADR(pParaArray));
			AdsEvent( 	Event 	:= TRUE);			
			IF NOT AdsEvent.Err AND_THEN Gvl.EventHandlingStatistic.CountIn(Status) //Add event to statistic and continue if added successfully
			THEN			
				State 										:= TCEVENTSTATE_SIGNALED;
			END_IF
		END_IF
	END_IF

(*****************************************************************)

END_FUNCTION_BLOCK

// POUs/Motion/TF5100-NCI/02_Options/Error/NciEventHandling
{attribute 'no_check'}
//EventHandlingGrp10 instance used inside
FUNCTION_BLOCK NciEventHandling
VAR CONSTANT
END_VAR                     								
VAR_INPUT                   								
	Enable													:	BOOL := TRUE; (* Show alarm message, warnings or hint. always reported !!! *)
	ConfirmTrig												:	BOOL := FALSE;
	SourceId												:	UDINT := 101200; //TwinCat-NCI channel default multisource Id + Channel id
	ErrorId													:	UDINT := 0;
	Name													:	STRING(30) := '';
	rNci													:	REFERENCE TO NCI_REF := 0;
END_VAR
VAR_OUTPUT
{attribute 'displaymode':='binary'}
	Status													:	DWORD;
	NoOfActiveEvents										:	INT;
END_VAR
VAR
(* Zwischenspeicher ***********************************************)
	QuitInternal 											: BOOL;

(* Timer **********************************************************)

(* Trigger ********************************************************)

(* Bausteine ******************************************************)
	Event													:	EventHandlingGrp10 := (
																	AutoConfirm			:= FALSE, 
																	SetClass 			:= TC2_SYSTEM.TCEVENTCLASS_ALARM );
	ChnEvent												:	NciChnEventHandling;

(* Dummy Speicher *************************************************)
	i														:	INT ;

END_VAR

(* Error message NCI channel to EventLogger 	V1.0	DS	*)
(***********************************************************)

(* Sequence **************************************************************)
IF __ISVALIDREF(rNci) 
THEN
	(* get Quit signal **************************************************)
	IF ConfirmTrig 
	THEN 
		QuitInternal 										:= TRUE; 
	END_IF (* set false see below *)

(* Event Logger Meldungen *****************************************************)
	Event.no[1].Flag 										:= rNci.IsEStopRequested;
	Event.no[2].Flag 										:= rNci.IsFeedFromBackupList;   
	Event.no[3].Flag 										:= rNci.IsMovingBackward;   
	
(*
	Event.no[4].Flag 										:= FALSE;
	Event.no[5].Flag 										:= FALSE;
	Event.no[6].Flag 										:= FALSE;
	Event.no[7].Flag 										:= FALSE;
	Event.no[8].Flag 										:= FALSE;
	Event.no[9].Flag 										:= FALSE;
	Event.no[10].Flag 										:= FALSE;
*)
(* workl Event Ctrl *************************************************)
	IF Event.no[1].Text2 <> Name OR Event.no[1].Text2 <> ''
	THEN
		//Init EventClass
		Event.no[1].eClass 									:= TC2_SYSTEM.TCEVENTCLASS_HINT;
		Event.no[2].eClass 									:= TC2_SYSTEM.TCEVENTCLASS_STATEINFO;
		Event.no[3].eClass 									:= TC2_SYSTEM.TCEVENTCLASS_STATEINFO;

		(* Init Name *)
		FOR i := Event.MIN_EVENT TO Event.MAX_EVENT DO
			Event.no[i].Text2								:= SEL(LEN(name)>1,CONCAT('Channel id:',DWORD_TO_STRING(rNci.NciToPlc.ChnId)),name);
		END_FOR
	END_IF

	Event(
		ConfirmTrig := ConfirmTrig,
		Disable		:= NOT Enable,
		SourceId	:= SourceId + rNci.NciToPlc.ChnId,
		Status	 	=> );	

(* Send ErrorId Message Text **********************************)
	ChnEvent(
		ConfirmTrig	:= NOT Enable OR QuitInternal OR ErrorId = 0 AND ChnEvent.State <> 0,
		Name		:= name,
		ChannelId	:= rNci.NciToPlc.ChnId,
		SourceId	:= Event.SourceId,
		Flag		:= ErrorId > 0 AND Enable,
		ErrorID		:= ErrorId,
		State		=> );

(* EventStatus *************************************************)
	Status													:= ChnEvent.Status OR Event.Status;
	NoOfActiveEvents										:= Event.NoOfActiveEvents + SEL(ChnEvent.Status.31 , 0, 1);

(* Error unkonw pointer or channel id *****************************)
ELSE
	NoOfActiveEvents										:= 0;
	ChnEvent(Flag := FALSE, ConfirmTrig := ChnEvent.State <> 0);
	Event(Disable := TRUE, Status =>  ); 
	Status													:= ChnEvent.Status OR Event.Status;
END_IF

(* Default reset Quit Internal *******************************)
	QuitInternal 											:= FALSE;

(**************************************************************)

METHOD PUBLIC confirm : bool  //Return value = TRUE if execution finished 
VAR_INPUT
END_VAR
QuitInternal 												:= TRUE;
confirm														:= TRUE;
END_METHOD

END_FUNCTION_BLOCK

// POUs/Motion/TF5100-NCI/02_Options/MFunctions/NciMFnc
{attribute 'no_check'}
FUNCTION_BLOCK NciMFnc
VAR_OUTPUT CONSTANT 
	MIN_M_FUNC												:	 UINT := 0;
	MAX_M_FUNC												:	 UINT := 159;
	
//Predefined M Functions
	M2_PRG_END												:	UINT := 2;
	M17_END_SUBROUTINE										:	UINT := 17;
	M30_PRG_END_WITH_ALL_MFUNC								:	UINT := 30; 
END_VAR                 									
VAR_INPUT               									
	ConfirmHsk												:	BOOL := FALSE; (* oder Methode benutzen *)
	FastMFuncReset											:	BOOL := FALSE; (* Signal Start Reser der unter FastMFuncNo angegebenen MFunc Nr. *)
	FastMFuncNo												:	UINT (MIN_M_FUNC..MAX_M_FUNC) := MIN_M_FUNC; (* Nr. der MFunktion die Resetet werden soll *)
	rNCIRef													:	REFERENCE TO NCI_REF := 0;
END_VAR                 									
VAR_OUTPUT              	
	HskReq													:	BOOL;
	HskId													:	UINT; 	
	CntActive												:	INT; //Count number of active M fucntions
	Active													:	BOOL; //Rising trigger M-Function active
	No														:	ARRAY[MIN_M_FUNC..MAX_M_FUNC] OF BOOL; (* Array of M-Functions *)
	rtNo													:	ARRAY[MIN_M_FUNC..MAX_M_FUNC] OF BOOL; (* rising trigger of M-Functions *)
END_VAR                     								
VAR
(* Zwischenspeicher ************************************************************)
	MemFnc													:	INT := -1;

(* Deklaration Trigger **********************************************************)

(* Zeiten ******************************************************************)

(* Bausteine ***************************************************************)
	ItpResetFastMFuncEx										:  ItpResetFastMFuncEx := (tTimeOut	:= DEFAULT_ADS_TIMEOUT);

(* Dummy Speicher **********************************************************)
	i														:	UINT := 0;
	OK														:	BOOL;
END_VAR

	(************************************************************************************)
	(*																					*)
	(*		B E C K H O F F   N E W   A U T O M A T I O N   T E C H N O L O G Y    		*)
	(*																					*)
	(*		Eiserstr.5	D-33415 Verl	Germany	phone:	+49-5246-0	www.Beckhoff.Com	*)
    (*																					*)
    (*		Bausteinbeschreibung	:	Auswerten von M-Funktionen						*)
	(*		TwinCAT-Version			:	2.11.x 											*)
	(*		Version					:	V2.0/ 05/20										*)
 	(*		Autor					:	Daniel Schlingmann								*)
	(*		Lib						:	TcNCI.Lib										*)
	(*																					*)
	(************************************************************************************)

(* evaluate M-function with additional acknowledge *********************************************************************)
	HskReq 													:= rNCIRef.NciToPlc.HskMFuncReq.0;
	HskId 													:= SEL(HskReq, 0, rNCIRef.NciToPlc.HskMFuncNo);

	(* Confirm request *)
	rNCIRef.PlcToNci.MFuncGranted.0 						:= (ConfirmHsk OR rNCIRef.PlcToNci.MFuncGranted.0) AND rNCIRef.NciToPlc.HskMFuncReq.0;

(* set all M-function setzen *)
	CntActive												:= 0;
	Active													:= FALSE;
	
	FOR i := MIN_M_FUNC TO MAX_M_FUNC DO
	 	OK	 												:= ItpIsFastMFunc(UINT_TO_INT(i),rNCIRef.NciToPlc) OR rNCIRef.NciToPlc.HskMFuncNo = i AND rNCIRef.NciToPlc.HskMFuncReq.0;
		rtNo[i]												:= NOT No[i] AND OK;
		No[i]												:= OK;
		IF No[i] 
		THEN 
			CntActive										:= CntActive + 1;		
			Active 											:= TRUE; 
		END_IF
	END_FOR

(* reset fast M-functions, ResetFastMFunc can also be used *)
	IF MemFnc < 0
	THEN
		IF FastMFuncReset
		THEN
			MemFnc 											:= 1;
			ResetFastMFunc(FastMFuncNo:= FastMFuncNo);
		END_IF
	ELSE 
		ResetFastMFunc(FastMFuncNo:= FastMFuncNo);		
	END_IF

(************************************************************************************)

METHOD PUBLIC confirm : BOOL //Return value = TRUE if execution finished
//required parameter
//rNCIRef
VAR_INPUT
END_VAR
IF __ISVALIDREF(rNCIRef)
THEN
	rNCIRef.PlcToNci.MFuncGranted.0 						:= rNCIRef.NciToPlc.HskMFuncReq.0;
	Confirm													:= NOT rNCIRef.NciToPlc.HskMFuncReq.0;
ELSE
	Confirm 												:= TRUE;
END_IF
END_METHOD

METHOD PUBLIC resetFastMFunc : BOOL //Return value = TRUE if busy
//required parameter
//rNCIRef
VAR_INPUT
	FastMFuncNo												:	UINT; (* number of M-function, which has to be resetted *)
END_VAR
IF NOT __ISVALIDREF(rNCIRef)
THEN
	ResetFastMFunc											:= FALSE;
	Return;	
END_IF

	IF ItpIsFastMFunc(UINT_TO_INT(FastMFuncNo),rNCIRef.NciToPlc) 
	THEN
		ItpResetFastMFuncEx.bExecute 						:= TRUE;
		MemFnc.0											:= TRUE;
	ELSIF NOT ItpResetFastMFuncEx.bBusy             		
	THEN                                            		
		ItpResetFastMFuncEx.bExecute 						:= FALSE;
	END_IF
	
	THIS^.FastMFuncNo										:= FastMFuncNo;

	ItpResetFastMFuncEx(
		bExecute	:= ,
		nMFuncNo	:= FastMFuncNo,
		tTimeOut	:= ,
		sNciToPlc	:= rNCIRef.NciToPlc,
		bBusy		=> ,
		bErr		=> ,
		nErrId	=> );
		
	IF NOT ItpResetFastMFuncEx.bBusy
	THEN
		IF ItpResetFastMFuncEx.bExecute
		THEN
			;
		//	Error											:=	ItpResetFastMFuncEx.bErr;
		//	ErrorId											:= ItpResetFastMFuncEx.nErrId;
		END_IF
		IF NOT ItpIsFastMFunc(UINT_TO_INT(FastMFuncNo),rNCIRef.NciToPlc) 
		THEN
			MemFnc											:= -1;
			ItpResetFastMFuncEx(bExecute := FALSE , sNciToPlc:= rNCIRef.NciToPlc);
		END_IF
	END_IF
	
	resetFastMFunc											:= ItpResetFastMFuncEx.bBusy;
END_METHOD

END_FUNCTION_BLOCK

// POUs/Motion/TF5100-NCI/02_Options/PlcItp/NciCreateItpTable
{attribute 'no_check'}
//Create Nci PlcInterpolation tabel
//
FUNCTION_BLOCK NciCreateItpTable
VAR_INPUT
	BlockNo													: UDINT := 0; //Block number addtional parameter for methods. At 0 -> block number will be automatically increased by every new entry
	OffsetFactorTblNumber									: UDINT := 100; 
	MaxTblNumber											: UDINT := 1000; 
END_VAR                     								
VAR_OUTPUT                  								
	Table													: ST_NciFeedGroupTable;
	FilledRows												: INT;
	LastBlockNo												: UDINT; //Last Blocknumber 
	Error													: BOOL;
{attribute 'displaymode':='hex'}
	ErrorID													: UDINT;
	ErrorText												: STRING(20);
END_VAR                     								
VAR
// Cache *******************************************
	TableNumber												: UDINT := 0;
	BlockCount												: UDINT := 1;

// Timer ******************************************************
// Trigger ****************************************************
// Blocks *****************************************************
	TblTemplate												: NciCreateItpTableEntryTemplate;
// Error ******************************************************
// Dummy Speicher *********************************************
	i														: INT := 0;
END_VAR

(* writing TcPlcInterpolation table				V1.5	*)
(********************************************************)

(* pleas use methods instead of the function-block body ********************)
	;
(***************************************************************************)

METHOD addCircleCIP : BOOL //Return value = TRUE if executed succesful
VAR_INPUT
	X														: LREAL := 0.0;
	Y														: LREAL := 0.0;
	Z														: LREAL := 0.0;
	Q1														: LREAL := 0.0;
	Q2														: LREAL := 0.0;
	Q3														: LREAL := 0.0;
	Q4														: LREAL := 0.0;
	Q5														: LREAL := 0.0;
	Velo													: LREAL; 	// mm/s 
	AccurateStop											: BOOL := FALSE;
	CIPPosX													: LREAL := 0.0;
	CIPPosY													: LREAL := 0.0;
	CIPPosZ													: LREAL := 0.0;
END_VAR
	(* NCI GeoCirclePlane schreiben									*)
	(*********************************************************)

(* Zielpos. in Tabelle schreiben ************************************************************)
	BlockCount 												:= BlockCount + 1;
	TblTemplate.GeoCircleCIP.nDisplayIndex := LastBlockNo 	:= SEL(BlockNo = 0, BlockNo, TableNumber * OffsetFactorTblNumber + BlockCount);
	TblTemplate.GeoCircleCIP.fEndPosX						:= X;
	TblTemplate.GeoCircleCIP.fEndPosY						:= Y;
	TblTemplate.GeoCircleCIP.fEndPosZ						:= Z;
	TblTemplate.GeoCircleCIP.fEndPosQ1						:= Q1;
	TblTemplate.GeoCircleCIP.fEndPosQ2						:= Q2;
	TblTemplate.GeoCircleCIP.fEndPosQ3						:= Q3;
	TblTemplate.GeoCircleCIP.fEndPosQ4						:= Q4;
	TblTemplate.GeoCircleCIP.fEndPosQ5						:= Q5;
	TblTemplate.GeoCircleCIP.fVelo							:= Velo;
	TblTemplate.GeoCircleCIP.bAccurateStop					:= AccurateStop;
	TblTemplate.GeoCircleCIP.fCIPPosX						:= CIPPosX;
	TblTemplate.GeoCircleCIP.fCIPPosY						:= CIPPosY;
	TblTemplate.GeoCircleCIP.fCIPPosZ						:= CIPPosZ;
                                                        	
	TblTemplate.InsertGeoCircleCIP(Table:= Table);    	
	Error													:= TblTemplate.Error;
	ErrorId													:= TblTemplate.ErrorId;
	ErrorText												:= TblTemplate.ErrorText;
	FilledRows												:= TblTemplate.FilledRows;

	AddCircleCip											:= NOT Error;
(***************************************************************************)
END_METHOD

METHOD addDwellTime : BOOL //Return value = TRUE if executed succesful
VAR_INPUT
	/// UCS ObjectID 
	Value													: LREAL ;
END_VAR
(*  													*)
(********************************************************)
	BlockCount 												:= BlockCount + 1;
	TblTemplate.DwellTime.nDisplayIndex	 := LastBlockNo 	:= SEL(BlockNo = 0, BlockNo, TableNumber * OffsetFactorTblNumber + BlockCount);
	TblTemplate.DwellTime.fDwellTime						:= Value;

	TblTemplate.InsertDwellTime(Table:= Table);
	Error													:= TblTemplate.Error;
	ErrorId													:= TblTemplate.ErrorId;
	ErrorText												:= TblTemplate.ErrorText;
	FilledRows												:= TblTemplate.FilledRows;

	AddDwellTime											:= not Error;	
	

(***************************************************************************)
END_METHOD

METHOD addEndOfTable : BOOL //Return value = TRUE if executed succesful
TblTemplate.InsertEndOfTable(Table:= Table);
Error													:= TblTemplate.Error;
ErrorId													:= TblTemplate.ErrorId;
ErrorText												:= TblTemplate.ErrorText;
FilledRows												:= TblTemplate.FilledRows;

AddEndOfTable											:= NOT Error;
END_METHOD

METHOD addMFuncFast : BOOL //Return value = TRUE if executed succesful
VAR_INPUT
	MFuncNo													: INT := 0;
END_VAR
(*														*)
(********************************************************)

(*************************************************************************************)
	BlockCount 												:= BlockCount + 1;
	TblTemplate.MFuncFast.nDisplayIndex := LastBlockNo 		:= SEL(BlockNo = 0, BlockNo, TableNumber * OffsetFactorTblNumber + BlockCount);
	TblTemplate.MFuncFast.nMFuncIn0							:= MFuncNo;
	TblTemplate.MFuncFast.nMFuncIn1							:= -1;
	TblTemplate.MFuncFast.nMFuncIn2							:= -1;
	TblTemplate.MFuncFast.nMFuncIn3							:= -1;
	TblTemplate.MFuncFast.nMFuncIn4							:= -1;
	TblTemplate.MFuncFast.nMFuncIn5							:= -1;
	TblTemplate.MFuncFast.nMFuncIn6							:= -1;
	TblTemplate.MFuncFast.nMFuncIn7							:= -1;
	
	TblTemplate.InsertMFuncFast(Table:= Table);
	Error													:= TblTemplate.Error;
	ErrorId													:= TblTemplate.ErrorId;
	ErrorText												:= TblTemplate.ErrorText;
	FilledRows												:= TblTemplate.FilledRows;
	
	AddMFuncFast											:= not Error;
(*************************************************************************************)
END_METHOD

METHOD addMFuncFastList : BOOL //Return value = TRUE if executed succesful
VAR_INPUT
	MFuncNo0												: INT := -1; //0-159 > Set to -1 to mark end of used MFunc
	MFuncNo1												: INT := -1; //0-159 > Set to -1 to mark end of used MFunc
	MFuncNo2												: INT := -1; //0-159 > Set to -1 to mark end of used MFunc
	MFuncNo3												: INT := -1; //0-159 > Set to -1 to mark end of used MFunc
	MFuncNo4												: INT := -1; //0-159 > Set to -1 to mark end of used MFunc
	MFuncNo5												: INT := -1; //0-159 > Set to -1 to mark end of used MFunc
	MFuncNo6												: INT := -1; //0-159 > Set to -1 to mark end of used MFunc
	MFuncNo7												: INT := -1; //0-159 > Set to -1 to mark end of used MFunc
END_VAR
(*														*)
(********************************************************)

(*************************************************************************************)
	BlockCount 												:= BlockCount + 1;
	TblTemplate.MFuncFast.nDisplayIndex := LastBlockNo 		:= SEL(BlockNo = 0, BlockNo, TableNumber * OffsetFactorTblNumber + BlockCount);
	TblTemplate.MFuncFast.nMFuncIn0							:= MFuncNo0;
	TblTemplate.MFuncFast.nMFuncIn1							:= MFuncNo1;
	TblTemplate.MFuncFast.nMFuncIn2							:= MFuncNo2;
	TblTemplate.MFuncFast.nMFuncIn3							:= MFuncNo3;
	TblTemplate.MFuncFast.nMFuncIn4							:= MFuncNo4;
	TblTemplate.MFuncFast.nMFuncIn5							:= MFuncNo5;
	TblTemplate.MFuncFast.nMFuncIn6							:= MFuncNo6;
	TblTemplate.MFuncFast.nMFuncIn7							:= MFuncNo7;
	
	TblTemplate.InsertMFuncFast(Table:= Table);
	Error													:= TblTemplate.Error;
	ErrorId													:= TblTemplate.ErrorId;
	ErrorText												:= TblTemplate.ErrorText;
	FilledRows												:= TblTemplate.FilledRows;
	
	AddMFuncFastList										:= NOT Error;
(*************************************************************************************)
END_METHOD

METHOD addMFuncHsk : BOOL //Return value = TRUE if executed succesful
VAR_INPUT
	MFuncNo													: INT := 0;
END_VAR
(* 														*)
(********************************************************)

(*************************************************************************************)
	BlockCount 												:= BlockCount + 1;
	TblTemplate.MFuncHsk.nDisplayIndex := LastBlockNo 		:= SEL(BlockNo = 0, BlockNo,  TableNumber * OffsetFactorTblNumber + BlockCount);
	TblTemplate.MFuncHsk.nMFunc								:= MFuncNo;
                                                        	
	TblTemplate.InsertMFuncHsk(Table:= Table);          	
	Error													:= TblTemplate.Error;
	ErrorId													:= TblTemplate.ErrorId;
	ErrorText												:= TblTemplate.ErrorText;
	FilledRows												:= TblTemplate.FilledRows;
	
	AddMFuncHsk												:= not Error;
(*************************************************************************************)
END_METHOD

METHOD addMFuncResetAllFast : BOOL //Return value = TRUE if executed succesful
VAR_INPUT
END_VAR
(* NCI ResetAllFastMFunc schreiben								*)
(*************************************************************************************)

(* confirmError all fast M-functions****************************************************)
	BlockCount 													:= BlockCount + 1;
	TblTemplate.MFuncResetAllFast.nDisplayIndex	:= LastBlockNo 	:= SEL(BlockNo = 0, BlockNo, TableNumber * OffsetFactorTblNumber + BlockCount);
	TblTemplate.InsertMFuncResetAllFast(Table:= Table);
	Error														:= TblTemplate.Error;
	ErrorId														:= TblTemplate.ErrorId;
	ErrorText													:= TblTemplate.ErrorText;
	FilledRows													:= TblTemplate.FilledRows;
	
	AddMFuncResetAllFast										:= not Error;
(*************************************************************************************)
END_METHOD

METHOD reset : BOOL //Return value = TRUE if execution finished
VAR_INPUT
END_VAR
TblTemplate.Reset(Table := Table);
FilledRows													:= 0;
BlockCount 													:= 0;
LastBlockNo													:= 0;
TableNumber 												:= TableNumber + 1;

IF TableNumber > MaxTblNumber 
THEN 
	TableNumber 											:= 1; 
END_IF

Error 														:= FALSE;
Errorid														:= 0;
ErrorText													:= '';
Reset														:= TRUE;
END_METHOD

METHOD setAxisDynamics : bool //Return value = TRUE if executed succesful
VAR_INPUT
	AxisNo													:	UDINT;
	Acc,Dec,Jerk											:	LREAL;
END_VAR
	(* NCI SetAxisDynamics schreiben						*)
	(*********************************************************)

(* Zielpos. in Tabelle schreiben ************************************************************)
	BlockCount 												:= BlockCount + 1;
	TblTemplate.AxisDynamics.nDisplayIndex := LastBlockNo := SEL(BlockNo = 0, BlockNo, TableNumber * OffsetFactorTblNumber + BlockCount);

	TblTemplate.AxisDynamics.nAxis 							:= AxisNo;
	TblTemplate.AxisDynamics.fDec							:= Dec;
	TblTemplate.AxisDynamics.fJerk							:= Jerk;
	TblTemplate.AxisDynamics.fAcc							:= Acc;
                                                        	
	TblTemplate.InsertAxisDynamics(Table:= Table);    	
	Error													:= TblTemplate.Error;
	ErrorId													:= TblTemplate.ErrorId;
	ErrorText												:= TblTemplate.ErrorText;
	FilledRows												:= TblTemplate.FilledRows;

	SetAxisDynamics											:= NOT Error;
(***************************************************************************)
END_METHOD

METHOD setBaseFrame : bool //Return value = TRUE if executed succesful
VAR_INPUT
    ShiftX													: LREAL;
    ShiftY													: LREAL;
    ShiftZ													: LREAL;
    RotX													: LREAL;
    RotY													: LREAL;
    RotZ													: LREAL;
    ShiftQ1													: LREAL;
    ShiftQ2													: LREAL;
    ShiftQ3													: LREAL;
    ShiftQ4													: LREAL;
    ShiftQ5													: LREAL;
END_VAR
	(* NCI SetBaseFrame schreiben						*)
	(*********************************************************)

(* Zielpos. in Tabelle schreiben ************************************************************)
	BlockCount 												:= BlockCount + 1;
	TblTemplate.BaseFrame.nDisplayIndex := LastBlockNo := SEL(BlockNo = 0, BlockNo, TableNumber * OffsetFactorTblNumber + BlockCount);

    TblTemplate.BaseFrame.fShiftX 							:= ShiftX;
    TblTemplate.BaseFrame.fShiftY							:= ShiftY;
    TblTemplate.BaseFrame.fShiftZ							:= ShiftZ;
    TblTemplate.BaseFrame.fRotX								:= RotX;
    TblTemplate.BaseFrame.fRotY								:= RotY;
    TblTemplate.BaseFrame.fRotZ								:= RotZ;
    TblTemplate.BaseFrame.fShiftQ1							:= ShiftQ1;
    TblTemplate.BaseFrame.fShiftQ2							:= ShiftQ2;
    TblTemplate.BaseFrame.fShiftQ3							:= ShiftQ3;
    TblTemplate.BaseFrame.fShiftQ4							:= ShiftQ4;
    TblTemplate.BaseFrame.fShiftQ5							:= ShiftQ5;
                       	
	TblTemplate.InsertBaseFrame(Table:= Table);    	
	Error													:= TblTemplate.Error;
	ErrorId													:= TblTemplate.ErrorId;
	ErrorText												:= TblTemplate.ErrorText;
	FilledRows												:= TblTemplate.FilledRows;

	SetBaseFrame											:= NOT Error;
(***************************************************************************)
END_METHOD

METHOD setCirclePlane : BOOL //Return value = TRUE if executed succesful
VAR_INPUT
	X														: LREAL := 0.0;
	Y														: LREAL := 0.0;
	Z														: LREAL := 0.0;
	Q1														: LREAL := 0.0;
	Q2														: LREAL := 0.0;
	Q3														: LREAL := 0.0;
	Q4														: LREAL := 0.0;
	Q5														: LREAL := 0.0;
	Velo													: LREAL; 	// mm/s 
	AccurateStop											: BOOL := FALSE;
	Clockwise												: BOOL := TRUE;
	Plane													: E_NciGeoPlane := E_NciGeoPlaneXY;
	CenterX													: LREAL := 0.0;
	CenterY													: LREAL := 0.0;
	CenterZ													: LREAL := 0.0;
END_VAR
	(* NCI GeoCirclePlane schreiben									*)
	(*********************************************************)

(* Zielpos. in Tabelle schreiben ************************************************************)
	BlockCount 												:= BlockCount + 1;
	TblTemplate.GeoCirclePlane.nDisplayIndex := LastBlockNo := SEL(BlockNo = 0, BlockNo, TableNumber * OffsetFactorTblNumber + BlockCount);
	TblTemplate.GeoCirclePlane.fEndPosX						:= X;
	TblTemplate.GeoCirclePlane.fEndPosY						:= Y;
	TblTemplate.GeoCirclePlane.fEndPosZ						:= Z;
	TblTemplate.GeoCirclePlane.fEndPosQ1					:= Q1;
	TblTemplate.GeoCirclePlane.fEndPosQ2					:= Q2;
	TblTemplate.GeoCirclePlane.fEndPosQ3					:= Q3;
	TblTemplate.GeoCirclePlane.fEndPosQ4					:= Q4;
	TblTemplate.GeoCirclePlane.fEndPosQ5					:= Q5;
	TblTemplate.GeoCirclePlane.fVelo						:= Velo;
	TblTemplate.GeoCirclePlane.bAccurateStop				:= AccurateStop;
	TblTemplate.GeoCirclePlane.bClockwise					:= Clockwise;
	TblTemplate.GeoCirclePlane.nPlane						:= Plane;
	TblTemplate.GeoCirclePlane.fCenterX						:= CenterX;
	TblTemplate.GeoCirclePlane.fCenterY						:= CenterY;
	TblTemplate.GeoCirclePlane.fCenterZ						:= CenterZ;
                                                        	
	TblTemplate.InsertGeoCirclePlane(Table:= Table);    	
	Error													:= TblTemplate.Error;
	ErrorId													:= TblTemplate.ErrorId;
	ErrorText												:= TblTemplate.ErrorText;
	FilledRows												:= TblTemplate.FilledRows;

	SetCirclePlane											:= NOT Error;
(***************************************************************************)
END_METHOD

METHOD setCoordinateSystem : BOOL //Return value = TRUE if executed succesful
VAR_INPUT
	/// UCS ObjectID 
	ObjectId												: UDINT := 0;
END_VAR
(* NCI UserKos schreiben															*)
(************************************************************************************)

(* User Koordinatensystem schreiben ************************************************************)
	BlockCount 												:= BlockCount + 1;
	TblTemplate.SetCoordinateSystem.nDisplayIndex := LastBlockNo := SEL(BlockNo = 0, BlockNo, TableNumber * OffsetFactorTblNumber + BlockCount);
	TblTemplate.SetCoordinateSystem.nObjectId				:= ObjectId;

	TblTemplate.InsertSetCoordinateSystem(Table:= Table);
	Error													:= TblTemplate.Error;
	ErrorId													:= TblTemplate.ErrorId;
	ErrorText												:= TblTemplate.ErrorText;
	FilledRows												:= TblTemplate.FilledRows;
	
	SetCoordinateSystem										:= not Error;
(*************************************************************************************)
END_METHOD

METHOD setDynOverride : BOOL //Return value = TRUE if executed succesful
VAR_INPUT
	/// UCS ObjectID 
	Value													: lreal := 0; //0.0-100.0%
END_VAR
(* NCI Oevrride schreiben											*)
(********************************************************************)

(* insert override **************************************************)
	(* apapt override *)
	BlockCount 												:= BlockCount + 1;
	TblTemplate.DynOverride.nDisplayIndex := LastBlockNo 		:= SEL(BlockNo = 0, BlockNo, TableNumber * OffsetFactorTblNumber + BlockCount);
	TblTemplate.DynOverride.fDynOvr								:= 0.01 * Value;

	TblTemplate.InsertDynOverride(Table:= Table);
	Error													:= TblTemplate.Error;
	ErrorId													:= TblTemplate.ErrorId;
	ErrorText												:= TblTemplate.ErrorText;
	FilledRows												:= TblTemplate.FilledRows;
	
	SetDynOverride											:= not Error;
(*************************************************************************************)
END_METHOD

METHOD setGeoBezier3 : booL //Return value = TRUE if executed succesful
VAR_INPUT
     ControlPoint1X											: LREAL;
     ControlPoint1Y											: LREAL;
     ControlPoint1Z											: LREAL;
     ControlPoint2X											: LREAL;
     ControlPoint2Y											: LREAL;
     ControlPoint2Z											: LREAL;
     EndPosX												: LREAL;
     EndPosY												: LREAL;
     EndPosZ												: LREAL;
     EndPosQ1												: LREAL;
     EndPosQ2												: LREAL;
     EndPosQ3												: LREAL;
     EndPosQ4												: LREAL;
     EndPosQ5												: LREAL;
     Velo													: LREAL;
     AccurateStop											: BOOL; (* VeloEnd := 0 *)
END_VAR
	(* NCI SetGeoBezier3 schreiben						*)
	(*********************************************************)

(* Zielpos. in Tabelle schreiben ************************************************************)
	BlockCount 												:= BlockCount + 1;
	TblTemplate.GeoBezier3.nDisplayIndex := LastBlockNo := SEL(BlockNo = 0, BlockNo, TableNumber * OffsetFactorTblNumber + BlockCount);

    TblTemplate.GeoBezier3.fControlPoint1X					:= ControlPoint1X;
    TblTemplate.GeoBezier3.fControlPoint1Y					:= ControlPoint1Y;
    TblTemplate.GeoBezier3.fControlPoint1Z					:= ControlPoint1Z;
    TblTemplate.GeoBezier3.fControlPoint2X					:= ControlPoint2X;
    TblTemplate.GeoBezier3.fControlPoint2Y					:= ControlPoint2Y;
    TblTemplate.GeoBezier3.fControlPoint2Z					:= ControlPoint2Z;
    TblTemplate.GeoBezier3.fEndPosX							:= EndPosX;
    TblTemplate.GeoBezier3.fEndPosY							:= EndPosY;
    TblTemplate.GeoBezier3.fEndPosZ							:= EndPosZ;
    TblTemplate.GeoBezier3.fEndPosQ1						:= EndPosQ1;
    TblTemplate.GeoBezier3.fEndPosQ2						:= EndPosQ2;
    TblTemplate.GeoBezier3.fEndPosQ3						:= EndPosQ3;
    TblTemplate.GeoBezier3.fEndPosQ4						:= EndPosQ4;
    TblTemplate.GeoBezier3.fEndPosQ5						:= EndPosQ5;
    TblTemplate.GeoBezier3.fVelo							:= Velo;
    TblTemplate.GeoBezier3.bAccurateStop					:= AccurateStop  ;                            	
	
	TblTemplate.InsertGeoBezier3(Table:= Table);    	
	Error													:= TblTemplate.Error;
	ErrorId													:= TblTemplate.ErrorId;
	ErrorText												:= TblTemplate.ErrorText;
	FilledRows												:= TblTemplate.FilledRows;

	SetGeoBezier3											:= NOT Error;
(***************************************************************************)
END_METHOD

METHOD setGeoBezier5 : booL //Return value = TRUE if executed succesful
VAR_INPUT
     ControlPoint1X											: LREAL;
     ControlPoint1Y											: LREAL;
     ControlPoint1Z											: LREAL;
     ControlPoint2X											: LREAL;
     ControlPoint2Y											: LREAL;
     ControlPoint2Z											: LREAL;
     ControlPoint3X											: LREAL;
     ControlPoint3Y											: LREAL;
     ControlPoint3Z											: LREAL;
     ControlPoint4X											: LREAL;
     ControlPoint4Y											: LREAL;
     ControlPoint4Z											: LREAL;
     EndPosX												: LREAL;
     EndPosY												: LREAL;
     EndPosZ												: LREAL;
     EndPosQ1												: LREAL;
     EndPosQ2												: LREAL;
     EndPosQ3												: LREAL;
     EndPosQ4												: LREAL;
     EndPosQ5												: LREAL;
     Velo													: LREAL;
     AccurateStop											: BOOL; (* VeloEnd := 0 *)
END_VAR
	(* NCI SetGeoBezier5 schreiben						*)
	(*********************************************************)

(* Zielpos. in Tabelle schreiben ************************************************************)
	BlockCount 												:= BlockCount + 1;
	TblTemplate.GeoBezier5.nDisplayIndex := LastBlockNo := SEL(BlockNo = 0, BlockNo, TableNumber * OffsetFactorTblNumber + BlockCount);

    TblTemplate.GeoBezier5.fControlPoint1X					:= ControlPoint1X;
    TblTemplate.GeoBezier5.fControlPoint1Y					:= ControlPoint1Y;
    TblTemplate.GeoBezier5.fControlPoint1Z					:= ControlPoint1Z;
    TblTemplate.GeoBezier5.fControlPoint2X					:= ControlPoint2X;
    TblTemplate.GeoBezier5.fControlPoint2Y					:= ControlPoint2Y;
    TblTemplate.GeoBezier5.fControlPoint2Z					:= ControlPoint2Z;
    TblTemplate.GeoBezier5.fControlPoint3X					:= ControlPoint3X;
    TblTemplate.GeoBezier5.fControlPoint3Y					:= ControlPoint3Y;
    TblTemplate.GeoBezier5.fControlPoint3Z					:= ControlPoint3Z;
    TblTemplate.GeoBezier5.fControlPoint4X					:= ControlPoint4X;
    TblTemplate.GeoBezier5.fControlPoint4Y					:= ControlPoint4Y;
    TblTemplate.GeoBezier5.fControlPoint4Z					:= ControlPoint4Z;
    TblTemplate.GeoBezier5.fEndPosX							:= EndPosX;
    TblTemplate.GeoBezier5.fEndPosY							:= EndPosY;
    TblTemplate.GeoBezier5.fEndPosZ							:= EndPosZ;
    TblTemplate.GeoBezier5.fEndPosQ1						:= EndPosQ1;
    TblTemplate.GeoBezier5.fEndPosQ2						:= EndPosQ2;
    TblTemplate.GeoBezier5.fEndPosQ3						:= EndPosQ3;
    TblTemplate.GeoBezier5.fEndPosQ4						:= EndPosQ4;
    TblTemplate.GeoBezier5.fEndPosQ5						:= EndPosQ5;
    TblTemplate.GeoBezier5.fVelo							:= Velo;
    TblTemplate.GeoBezier5.bAccurateStop					:= AccurateStop  ;                            	
	
	TblTemplate.InsertGeoBezier5(Table:= Table);    	
	Error													:= TblTemplate.Error;
	ErrorId													:= TblTemplate.ErrorId;
	ErrorText												:= TblTemplate.ErrorText;
	FilledRows												:= TblTemplate.FilledRows;

	SetGeoBezier5											:= NOT Error;
(***************************************************************************)
END_METHOD

METHOD setGeoLine : BOOL //Return value = TRUE if executed succesful
VAR_INPUT
	X														: LREAL := 0.0;
	Y														: LREAL := 0.0;
	Z														: LREAL := 0.0;
	Q1														: LREAL := 0.0;
	Q2														: LREAL := 0.0;
	Q3														: LREAL := 0.0;
	Q4														: LREAL := 0.0;
	Q5														: LREAL := 0.0;
	Velo													: LREAL; 	// mm/s 
	AccurateStop											: BOOL := FALSE;
END_VAR
(* writing NCI GeoLine 									*)
(********************************************************)

(***************************************************************************)
	BlockCount 												:= BlockCount + 1;
	TblTemplate.GeoLine.nDisplayIndex := LastBlockNo 		:= SEL(BlockNo = 0, BlockNo, TableNumber * OffsetFactorTblNumber + BlockCount);
	TblTemplate.GeoLine.fEndPosX							:= X;
	TblTemplate.GeoLine.fEndPosY							:= Y;
	TblTemplate.GeoLine.fEndPosZ							:= Z;
	TblTemplate.GeoLine.fEndPosQ1							:= Q1 ;
	TblTemplate.GeoLine.fEndPosQ2							:= Q2;
	TblTemplate.GeoLine.fEndPosQ3							:= Q3;
	TblTemplate.GeoLine.fEndPosQ4							:= Q4;
	TblTemplate.GeoLine.fEndPosQ5							:= Q5;
	TblTemplate.GeoLine.fVelo								:= Velo;
	TblTemplate.GeoLine.bRapidTraverse						:= Velo = 0.0;
	TblTemplate.GeoLine.bAccurateStop						:= AccurateStop;
                                                        	
	TblTemplate.InsertGeoLine(Table:= Table);           	
	Error													:= TblTemplate.Error;
	ErrorId													:= TblTemplate.ErrorId;
	ErrorText												:= TblTemplate.ErrorText;
	FilledRows												:= TblTemplate.FilledRows;
	
	SetGeoLine												:= not Error;
(***************************************************************************)
END_METHOD

METHOD setGeoStart : BOOL //Return value = TRUE if executed succesful
VAR_INPUT
	X														: LREAL := 0.0;
	Y														: LREAL := 0.0;
	Z														: LREAL := 0.0;
	Q1														: LREAL := 0.0;
	Q2														: LREAL := 0.0;
	Q3														: LREAL := 0.0;
	Q4														: LREAL := 0.0;
	Q5														: LREAL := 0.0;
END_VAR
(* writing NCI GeoLine 									*)
(********************************************************)

(***************************************************************************)
	TblTemplate.GeoStart.fPosX								:= X;
	TblTemplate.GeoStart.fPosY								:= Y;
	TblTemplate.GeoStart.fPosZ								:= Z;
	TblTemplate.GeoStart.fPosQ1								:= Q1 ;
	TblTemplate.GeoStart.fPosQ2								:= Q2;
	TblTemplate.GeoStart.fPosQ3								:= Q3;
	TblTemplate.GeoStart.fPosQ4								:= Q4;
	TblTemplate.GeoStart.fPosQ5								:= Q5;
                                                        	
	TblTemplate.InsertGeoStart(Table:= Table);           	
	Error													:= TblTemplate.Error;
	ErrorId													:= TblTemplate.ErrorId;
	ErrorText												:= TblTemplate.ErrorText;
	FilledRows												:= TblTemplate.FilledRows;
	
	SetGeoStart												:= not Error;
(***************************************************************************)
END_METHOD

METHOD setHParam : booL //Return value = TRUE if executed succesful
VAR_INPUT
	HParam													: UDINT;
END_VAR
(* 														*)
(********************************************************)

(*************************************************************************************)
	BlockCount 												:= BlockCount + 1;
	TblTemplate.HParam.nDisplayIndex := LastBlockNo 		:= SEL(BlockNo = 0, BlockNo,  TableNumber * OffsetFactorTblNumber + BlockCount);
	TblTemplate.HParam.nHParam								:= HParam;
                                                        	
	TblTemplate.InsertHParam(Table:= Table);          	
	Error													:= TblTemplate.Error;
	ErrorId													:= TblTemplate.ErrorId;
	ErrorText												:= TblTemplate.ErrorText;
	FilledRows												:= TblTemplate.FilledRows;
	
	SetHParam												:= NOT Error;
(*************************************************************************************)
END_METHOD

METHOD setPathDynamics : BOOL //Return value = TRUE if executed succesful
VAR_INPUT
	Acc,Dec,Jerk											:	LREAL;
END_VAR
	(* NCI SetPathDynamics schreiben						*)
	(*********************************************************)

(* Zielpos. in Tabelle schreiben ************************************************************)
	BlockCount 												:= BlockCount + 1;
	TblTemplate.PathDynamics.nDisplayIndex := LastBlockNo := SEL(BlockNo = 0, BlockNo, TableNumber * OffsetFactorTblNumber + BlockCount);

	TblTemplate.PathDynamics.fDec							:= Dec;
	TblTemplate.PathDynamics.fJerk							:= Jerk;
	TblTemplate.PathDynamics.fAcc							:= Acc;
                                                        	
	TblTemplate.InsertPathDynamics(Table:= Table);    	
	Error													:= TblTemplate.Error;
	ErrorId													:= TblTemplate.ErrorId;
	ErrorText												:= TblTemplate.ErrorText;
	FilledRows												:= TblTemplate.FilledRows;

	SetPathDynamics											:= NOT Error;
(***************************************************************************)
END_METHOD

METHOD setSParam : bool //Return value = TRUE if executed succesful
VAR_INPUT
	SParam													: UINT;
END_VAR
(* 														*)
(********************************************************)

(*************************************************************************************)
	BlockCount 												:= BlockCount + 1;
	TblTemplate.SParam.nDisplayIndex := LastBlockNo 		:= SEL(BlockNo = 0, BlockNo,  TableNumber * OffsetFactorTblNumber + BlockCount);
	TblTemplate.SParam.nSParam								:= SParam;
                                                        	
	TblTemplate.InsertSParam(Table:= Table);          	
	Error													:= TblTemplate.Error;
	ErrorId													:= TblTemplate.ErrorId;
	ErrorText												:= TblTemplate.ErrorText;
	FilledRows												:= TblTemplate.FilledRows;
	
	SetSParam												:= NOT Error;
(*************************************************************************************)
END_METHOD

METHOD setTangFollowingDesc : booL //Return value = TRUE if executed succesful
VAR_INPUT
    TangOn													: BOOL;
    TangAxis												: E_NciAxesInGroup;  
    PathAxis1												: E_NciAxesInGroup; 
    PathAxis2												: E_NciAxesInGroup; 
    Offset													: LREAL; 
    CriticalAngle1											: LREAL;
    TfBehavior												: E_TangentialFollowingBehavior; 
END_VAR
	(* NCI SetTangFollowingDesc schreiben						*)
	(*********************************************************)

(* Zielpos. in Tabelle schreiben ************************************************************)
	BlockCount 												:= BlockCount + 1;
	LastBlockNo 											:= SEL(BlockNo = 0, BlockNo, TableNumber * OffsetFactorTblNumber + BlockCount);

    TblTemplate.TangentialFollowingDesc.bTangOn				:= TangOn;
    TblTemplate.TangentialFollowingDesc.nTangAxis			:= TangAxis;
    TblTemplate.TangentialFollowingDesc.nPathAxis1			:= PathAxis1;
    TblTemplate.TangentialFollowingDesc.nPathAxis2			:= PathAxis2;
    TblTemplate.TangentialFollowingDesc.fOffset				:= Offset;
    TblTemplate.TangentialFollowingDesc.fCriticalAngle1		:= CriticalAngle1;
    TblTemplate.TangentialFollowingDesc.nTfBehavior			:= TfBehavior;
                       	
	TblTemplate.InsertTangFollowingDesc(Table:= Table);    	
	Error													:= TblTemplate.Error;
	ErrorId													:= TblTemplate.ErrorId;
	ErrorText												:= TblTemplate.ErrorText;
	FilledRows												:= TblTemplate.FilledRows;

	SetTangFollowingDesc									:= NOT Error;
(***************************************************************************)
END_METHOD

METHOD setTParam : bool //Return value = TRUE if executed succesful
VAR_INPUT
	TParam													: UINT;
END_VAR
(* 														*)
(********************************************************)

(*************************************************************************************)
	BlockCount 												:= BlockCount + 1;
	TblTemplate.TParam.nDisplayIndex := LastBlockNo 		:= SEL(BlockNo = 0, BlockNo,  TableNumber * OffsetFactorTblNumber + BlockCount);
	TblTemplate.TParam.nTParam								:= TParam;
                                                        	
	TblTemplate.InsertTParam(Table:= Table);          	
	Error													:= TblTemplate.Error;
	ErrorId													:= TblTemplate.ErrorId;
	ErrorText												:= TblTemplate.ErrorText;
	FilledRows												:= TblTemplate.FilledRows;
	
	SetTParam												:= NOT Error;
(**************************************************************************)
END_METHOD

METHOD setVertexSmoothing : BOOL //Return value = TRUE if executed succesful
VAR_INPUT
	Radius													: LREAL := 0.0;
	VertSmType												: UDINT := 5;
	VertSmSubType											: UDINT := 3;
END_VAR
(* writing NCI Vertex smoothing 								*)
(****************************************************************)

(* writing into table	*****************************************)
	BlockCount 												:= BlockCount + 1;
	TblTemplate.VertexSmoothing.nDisplayIndex := LastBlockNo := SEL(BlockNo = 0, BlockNo, TableNumber * OffsetFactorTblNumber + BlockCount);
	TblTemplate.VertexSmoothing.nType						:= VertSmType;
	TblTemplate.VertexSmoothing.nSubtype					:= VertSmSubtype; (* 	1: constant radius tolerance
																					2: distance between Abstand intersectoin point and peal point
																					3: adaptiv raidus tolerance
																					*)
	TblTemplate.VertexSmoothing.fRadius						:= Radius; (* mm *)

	TblTemplate.InsertVertexSmoothing(Table:= Table);
	Error													:= TblTemplate.Error;
	ErrorId													:= TblTemplate.ErrorId;
	ErrorText												:= TblTemplate.ErrorText;
	FilledRows												:= TblTemplate.FilledRows;
	SetVertexSmoothing										:= not Error;
(*************************************************************************************)
END_METHOD

END_FUNCTION_BLOCK

// POUs/Motion/TF5100-NCI/02_Options/PlcItp/NciCreateItpTableEntryTemplate
FUNCTION_BLOCK NciCreateItpTableEntryTemplate
VAR_INPUT
	EndOfTables												: ST_NciEndOfTables;
	GeoCirclePlane											: ST_NciGeoCirclePlane;
	GeoCircleCIP											: ST_NciGeoCircleCIP;
	GeoLine													: ST_NciGeoLine;
	GeoBezier3												: ST_NciGeoBezier3;
	GeoBezier5												: ST_NciGeoBezier5;	
	GeoStart												: ST_NciGeoStart;
	TangentialFollowingDesc									: ST_NciTangentialFollowingDesc;
	MFuncHsk												: ST_NciMFuncHsk;
	MFuncFast												: ST_NciMFuncFast;
	MFuncResetAllFast										: ST_NciMFuncResetAllFast;
	HParam													: ST_NciHParam;
	SParam													: ST_NciSParam;
	TParam													: ST_NciTParam;
	DynOverride												: ST_NciDynOvr;
	VertexSmoothing											: ST_NciVertexSmoothing;
	PathDynamics											: ST_NciPathDynamics;
	BaseFrame												: ST_NciBaseFrame;
	SetCoordinateSystem										: ST_NciSetCoordinateSystem;
	AxisDynamics											: ST_NciAxisDynamics;
	DwellTime												: ST_NciDwellTime;
END_VAR
VAR_OUTPUT
	FilledRows												: INT;
	Error													: BOOL;
{attribute 'displaymode':='hex'}
	ErrorId													: UDINT;
	ErrorText												: STRING(20);
END_VAR                 									
VAR                     									
	TblPrep													: FB_NciFeedTablePreparation;
END_VAR

(* NCI Table entry template				 	V2.0	*)
(****************************************************)

(******************************************************************************)
;
(******************************************************************************)

METHOD insertAxisDynamics : bool //Return value = TRUE if executed succesful
VAR_IN_OUT
	Table													: ST_NciFeedGroupTable;
END_VAR
	TblPrep(
		nEntryType			:= AxisDynamics.nEntryType,
		pEntry				:= ADR(AxisDynamics),
		stFeedGroupTable	:= Table,
		nFilledRows			=> FilledRows,
		bError				=> ,
		nErrorId			=> );

	IF TblPrep.bError 
	THEN
		Error												:= TRUE;
		ErrorText											:= CONCAT('AxisDynamics - JobNo. :',UDINT_TO_STRING(AxisDynamics.nDisplayIndex));
		ErrorId												:= TblPrep.nErrorId;
	ELSE
		insertAxisDynamics									:= TRUE;
	END_IF
END_METHOD

METHOD insertBaseFrame : bool //Return value = TRUE if executed succesful
VAR_IN_OUT
	Table													: ST_NciFeedGroupTable;
END_VAR
	TblPrep(
		nEntryType		:= BaseFrame.nEntryType,
		pEntry			:= ADR(BaseFrame),
		stFeedGroupTable:= Table,
		nFilledRows		=> FilledRows,
		bError			=> ,
		nErrorId		=> );

	IF TblPrep.bError 
	THEN
		Error												:= TRUE;
		ErrorText											:= CONCAT('BaseFrame - JobNo. :',UDINT_TO_STRING(BaseFrame.nDisplayIndex));
		ErrorId												:= TblPrep.nErrorId;
	ELSE
		insertBaseFrame										:= TRUE;
	END_IF
END_METHOD

METHOD insertDwellTime : booL //Return value = TRUE if executed succesful
VAR_IN_OUT
	Table													: ST_NciFeedGroupTable;
END_VAR
	TblPrep(
		nEntryType		:= DwellTime.nEntryType,
		pEntry			:= ADR(DwellTime),
		stFeedGroupTable:= Table,
		nFilledRows		=> FilledRows,
		bError			=> ,
		nErrorId		=> );

	IF TblPrep.bError 
	THEN
		Error												:= TRUE;
		ErrorText											:= CONCAT('DwellTime - JobNo. :',UDINT_TO_STRING(DwellTime.nDisplayIndex));
		ErrorId												:= TblPrep.nErrorId;
	ELSE
		insertDwellTime										:= TRUE;
	END_IF
END_METHOD

METHOD insertDynOverride : booL //Return value = TRUE if executed succesful
VAR_IN_OUT
	Table													: ST_NciFeedGroupTable;
END_VAR
	TblPrep(
		nEntryType			:= DynOverride.nEntryType,
		pEntry				:= ADR(DynOverride),
		stFeedGroupTable	:= Table,
		nFilledRows			=> FilledRows,
		bError				=> ,
		nErrorId			=> );

	IF TblPrep.bError THEN
		Error												:= TRUE;
		ErrorText											:= CONCAT('DynOverride - JobNo. :',UDINT_TO_STRING(DynOverride.nDisplayIndex));
		ErrorId												:= TblPrep.nErrorId;
	ELSE
		insertDynOverride									:= TRUE;
	END_IF
END_METHOD

METHOD insertEndOfTable : bool //Return value = TRUE if executed succesful
VAR_IN_OUT
	Table													: ST_NciFeedGroupTable;
END_VAR
	TblPrep(
		nEntryType			:= EndOfTables.nEntryType,
		pEntry				:= ADR(EndOfTables),
		stFeedGroupTable	:= Table,
		nFilledRows			=> FilledRows,
		bError				=> ,
		nErrorId			=> );

	IF TblPrep.bError THEN
		Error												:= TRUE;
		ErrorText											:= CONCAT('EndOfTables - FilledRows :',INT_TO_STRING(FilledRows));
		ErrorId												:= TblPrep.nErrorId;
	ELSE
		insertEndOfTable									:= TRUE;
	END_IF
END_METHOD

METHOD insertGeoBezier3 : booL //Return value = TRUE if executed succesful
VAR_IN_OUT
	Table													: ST_NciFeedGroupTable;
END_VAR
	TblPrep(
		nEntryType			:= GeoBezier3.nEntryType,
		pEntry				:= ADR(GeoBezier3),
		stFeedGroupTable	:= Table,
		nFilledRows			=> FilledRows,
		bError				=> ,
		nErrorId			=> );

	IF TblPrep.bError THEN
		Error												:= TRUE;
		ErrorText											:= CONCAT('GeoBezier3 - JobNo. :',UDINT_TO_STRING(GeoBezier3.nDisplayIndex));
		ErrorId												:= TblPrep.nErrorId;
	ELSE
		insertGeoBezier3									:= TRUE;
	END_IF
END_METHOD

METHOD insertGeoBezier5 : booL //Return value = TRUE if executed succesful
VAR_IN_OUT
	Table													: ST_NciFeedGroupTable;
END_VAR
	TblPrep(
		nEntryType			:= GeoBezier5.nEntryType,
		pEntry				:= ADR(GeoBezier5),
		stFeedGroupTable	:= Table,
		nFilledRows			=> FilledRows,
		bError				=> ,
		nErrorId			=> );

	IF TblPrep.bError THEN
		Error												:= TRUE;
		ErrorText											:= CONCAT('GeoBezier5 - JobNo. :',UDINT_TO_STRING(GeoBezier5.nDisplayIndex));
		ErrorId												:= TblPrep.nErrorId;
	ELSE
		insertGeoBezier5									:= TRUE;
	END_IF
END_METHOD

METHOD insertGeoCircleCIP : booL //Return value = TRUE if executed succesful
VAR_IN_OUT
	Table													: ST_NciFeedGroupTable;
END_VAR
	TblPrep(
		nEntryType			:= GeoCircleCIP.nEntryType,
		pEntry				:= ADR(GeoCircleCIP),
		stFeedGroupTable	:= Table,
		nFilledRows			=> FilledRows,
		bError				=> ,
		nErrorId			=> );

	IF TblPrep.bError 
	THEN
		Error												:= TRUE;
		ErrorText											:= CONCAT('GeoCircleCIP - JobNo. :',UDINT_TO_STRING(GeoCirclePlane.nDisplayIndex));
		ErrorId												:= TblPrep.nErrorId;
	ELSE
		insertGeoCircleCIP									:= TRUE;
	END_IF
END_METHOD

METHOD insertGeoCirclePlane : BOOL //Return value = TRUE if executed succesful
VAR_IN_OUT
	Table													: ST_NciFeedGroupTable;
END_VAR
	TblPrep(
		nEntryType			:= GeoCirclePlane.nEntryType,
		pEntry				:= ADR(GeoCirclePlane),
		stFeedGroupTable	:= Table,
		nFilledRows			=> FilledRows,
		bError				=> ,
		nErrorId			=> );

	IF TblPrep.bError 
	THEN
		Error												:= TRUE;
		ErrorText											:= CONCAT('GeoCirclePlane - JobNo. :',UDINT_TO_STRING(GeoCirclePlane.nDisplayIndex));
		ErrorId												:= TblPrep.nErrorId;
	ELSE
		insertGeoCirclePlane								:= TRUE;
	END_IF
END_METHOD

METHOD insertGeoLine : boOL //Return value = TRUE if executed succesful
VAR_IN_OUT
	Table													: ST_NciFeedGroupTable;
END_VAR
	TblPrep(
		nEntryType			:= GeoLine.nEntryType,
		pEntry				:= ADR(GeoLine),
		stFeedGroupTable	:= Table,
		nFilledRows			=> FilledRows,
		bError				=> ,
		nErrorId			=> );

	IF TblPrep.bError 
	THEN
		Error												:= TRUE;
		ErrorText											:= CONCAT('GeoLine - JobNo. :',UDINT_TO_STRING(GeoLine.nDisplayIndex));
		ErrorId												:= TblPrep.nErrorId;
	ELSE
		insertGeoLine										:= TRUE;
	END_IF
END_METHOD

METHOD insertGeoStart : booL //Return value = TRUE if executed succesful
VAR_IN_OUT
	Table													: ST_NciFeedGroupTable;
END_VAR
	TblPrep(
		nEntryType			:= GeoStart.nEntryType,
		pEntry				:= ADR(GeoStart),
		stFeedGroupTable	:= Table,
		nFilledRows			=> FilledRows,
		bError				=> ,
		nErrorId			=> );

	IF TblPrep.bError 
	THEN
		Error												:= TRUE;
		ErrorText											:= CONCAT('GeoStart - FilledRows. :',INT_TO_STRING(FilledRows));
		ErrorId												:= TblPrep.nErrorId;
	ELSE
		insertGeoStart										:= TRUE;
	END_IF
END_METHOD

METHOD insertHParam : booL //Return value = TRUE if executed succesful
VAR_IN_OUT
	Table													: ST_NciFeedGroupTable;
END_VAR
	TblPrep(
		nEntryType			:= HParam.nEntryType,
		pEntry				:= ADR(HParam),
		stFeedGroupTable	:= Table,
		nFilledRows			=> FilledRows,
		bError				=> ,
		nErrorId			=> );

	IF TblPrep.bError 
	THEN
		Error												:= TRUE;
		ErrorText											:= CONCAT('HParam - JobNo. :',UDINT_TO_STRING(HParam.nDisplayIndex));
		ErrorId												:= TblPrep.nErrorId;
	ELSE
		insertHParam										:= TRUE;
	END_IF
END_METHOD

METHOD insertMFuncFast : booL //Return value = TRUE if executed succesful
VAR_IN_OUT
	Table													: ST_NciFeedGroupTable;
END_VAR
	TblPrep(
		nEntryType			:= MFuncFast.nEntryType,
		pEntry				:= ADR(MFuncFast),
		stFeedGroupTable	:= Table,
		nFilledRows			=> FilledRows,
		bError				=> ,
		nErrorId			=> );

	IF TblPrep.bError 
	THEN
		Error												:= TRUE;
		ErrorText											:= CONCAT('MFuncFastList - JobNo. :',UDINT_TO_STRING(MFuncFast.nDisplayIndex));
		ErrorId												:= TblPrep.nErrorId;
	ELSE
		insertMFuncFast										:= TRUE;
	END_IF
END_METHOD

METHOD insertMFuncHsk : bool //Return value = TRUE if executed succesful
VAR_IN_OUT
	Table													: ST_NciFeedGroupTable;
END_VAR
	TblPrep(
		nEntryType			:= MFuncHsk.nEntryType,
		pEntry				:= ADR(MFuncHsk),
		stFeedGroupTable	:= Table,
		nFilledRows			=> FilledRows,
		bError				=> ,
		nErrorId			=> );

	IF TblPrep.bError 
	THEN
		Error												:= TRUE;
		ErrorText											:= CONCAT('MFuncHsk - JobNo. :',UDINT_TO_STRING(MFuncHsk.nDisplayIndex));
		ErrorId												:= TblPrep.nErrorId;
	ELSE
		insertMFuncHsk										:= TRUE;
	END_IF
END_METHOD

METHOD insertMFuncResetAllFast : bool //Return value = TRUE if executed succesful
VAR_IN_OUT
	Table													: ST_NciFeedGroupTable;
END_VAR
	TblPrep(
		nEntryType			:= MFuncResetAllFast.nEntryType,
		pEntry				:= ADR(MFuncResetAllFast),
		stFeedGroupTable	:= Table,
		nFilledRows			=> FilledRows,
		bError				=> ,
		nErrorId			=> );

	IF TblPrep.bError 
	THEN
		Error												:= TRUE;
		ErrorText											:= CONCAT('MFuncResetAllFast - JobNo. :',UDINT_TO_STRING(MFuncResetAllFast.nDisplayIndex));
		ErrorId												:= TblPrep.nErrorId;
	ELSE
		insertMFuncResetAllFast								:= TRUE;
	END_IF
END_METHOD

METHOD insertPathDynamics : BOOL //Return value = TRUE if executed succesful
VAR_IN_OUT
	Table													: ST_NciFeedGroupTable;
END_VAR
	TblPrep(
		nEntryType			:= PathDynamics.nEntryType,
		pEntry				:= ADR(PathDynamics),
		stFeedGroupTable	:= Table,
		nFilledRows			=> FilledRows,
		bError				=> ,
		nErrorId			=> );

	IF TblPrep.bError 
	THEN
		Error												:= TRUE;
		ErrorText											:= CONCAT('PathDynamics - JobNo. :',UDINT_TO_STRING(PathDynamics.nDisplayIndex));
		ErrorId												:= TblPrep.nErrorId;
	ELSE
		insertPathDynamics									:= TRUE;
	END_IF
END_METHOD

METHOD insertSetCoordinateSystem : bool //Return value = TRUE if executed succesful
VAR_IN_OUT
	Table													: ST_NciFeedGroupTable;
END_VAR
	TblPrep(
		nEntryType			:= SetCoordinateSystem.nEntryType,
		pEntry				:= ADR(SetCoordinateSystem),
		stFeedGroupTable	:= Table,
		nFilledRows			=> FilledRows,
		bError				=> ,
		nErrorId			=> );

	IF TblPrep.bError 
	THEN
		Error												:= TRUE;
		ErrorText											:= CONCAT('SetCoordinateSystem - JobNo. :',UDINT_TO_STRING(SetCoordinateSystem.nDisplayIndex));
		ErrorId												:= TblPrep.nErrorId;
	ELSE
		insertSetCoordinateSystem							:= TRUE;
	END_IF
END_METHOD

METHOD insertSParam : bool //Return value = TRUE if executed succesful
VAR_IN_OUT
	Table													: ST_NciFeedGroupTable;
END_VAR
	TblPrep(
		nEntryType			:= SParam.nEntryType,
		pEntry				:= ADR(SParam),
		stFeedGroupTable	:= Table,
		nFilledRows			=> FilledRows,
		bError				=> ,
		nErrorId			=> );

	IF TblPrep.bError 
	THEN
		Error												:= TRUE;
		ErrorText											:= CONCAT('SParam - JobNo. :',UDINT_TO_STRING(SParam.nDisplayIndex));
		ErrorId												:= TblPrep.nErrorId;
	ELSE
		insertSParam										:= TRUE;
	END_IF
END_METHOD

METHOD insertTangFollowingDesc : booL //Return value = TRUE if executed succesful
VAR_IN_OUT
	Table													: ST_NciFeedGroupTable;
END_VAR
	TblPrep(
		nEntryType			:= TangentialFollowingDesc.nEntryType,
		pEntry				:= ADR(TangentialFollowingDesc),
		stFeedGroupTable	:= Table,
		nFilledRows			=> FilledRows,
		bError				=> ,
		nErrorId			=> );

	IF TblPrep.bError 
	THEN
		Error												:= TRUE;
		ErrorText											:= CONCAT('TangentialFollowingDesc - JobNo. :','~');
		ErrorId												:= TblPrep.nErrorId;
	ELSE
		insertTangFollowingDesc								:= TRUE;
	END_IF
END_METHOD

METHOD insertTParam : bool //Return value = TRUE if executed succesful
VAR_IN_OUT
	Table													: ST_NciFeedGroupTable;
END_VAR
	TblPrep(
		nEntryType			:= TParam.nEntryType,
		pEntry				:= ADR(TParam),
		stFeedGroupTable	:= Table,
		nFilledRows			=> FilledRows,
		bError				=> ,
		nErrorId			=> );

	IF TblPrep.bError 
	THEN
		Error												:= TRUE;
		ErrorText											:= CONCAT('TParam - JobNo. :',UDINT_TO_STRING(TParam.nDisplayIndex));
		ErrorId												:= TblPrep.nErrorId;
	ELSE
		insertTParam										:= TRUE;
	END_IF
END_METHOD

METHOD insertVertexSmoothing : BOOL //Return value = TRUE if executed succesful
VAR_IN_OUT
	Table													: ST_NciFeedGroupTable;
END_VAR
	TblPrep(
		nEntryType			:= VertexSmoothing.nEntryType,
		pEntry				:= ADR(VertexSmoothing),
		stFeedGroupTable	:= Table,
		nFilledRows			=> FilledRows,
		bError				=> ,
		nErrorId			=> );

	IF TblPrep.bError 
	THEN
		Error												:= TRUE;
		ErrorText											:= CONCAT('VertexSmoothing - JobNo. :',UDINT_TO_STRING(VertexSmoothing.nDisplayIndex));
		ErrorId												:= TblPrep.nErrorId;
	ELSE
		insertVertexSmoothing								:= TRUE;
	END_IF
END_METHOD

METHOD reset : BOOL  //Return value = TRUE if execution finished
VAR_IN_OUT
	Table													: ST_NciFeedGroupTable;
END_VAR
TblPrep(
	nEntryType			:= ,
	pEntry				:= ,
	bResetTable			:= TRUE,
	bResetAll			:= TRUE,
	stFeedGroupTable	:= Table,
	nFilledRows			=> FilledRows,
	bError				=> ,
	nErrorId			=> );

TblPrep.bResetTable											:= FALSE;
TblPrep.bResetAll											:= FALSE;
Error														:= FALSE;
ErrorText													:= '';
ErrorId														:= 0;
Reset														:= TRUE;
END_METHOD

END_FUNCTION_BLOCK

// POUs/Motion/TF511x-KIN/03_DUTs/Trafo/UCS
{attribute 'hide'}
FUNCTION_BLOCK UCS
VAR_INPUT
	oid														:	UDINT := 0;		//Object identifier
	vTranslation 											:	VECTOR;
 	vRotation 												:	VECTOR;
	Valid													:	BOOL := FALSE;
END_VAR
VAR_OUTPUT
END_VAR
VAR
END_VAR

METHOD delete : BOOL
VAR_INPUT
END_VAR
MEMSET(ADR(vTranslation),0,SIZEOF(vTranslation));
MEMSET(ADR(VRotation),0,SIZEOF(VRotation));
oid 													:= 0;
delete	:= TRUE;
END_METHOD

END_FUNCTION_BLOCK

// POUs/Motion/TF5100-NCI/02_Options/RParameter/NCiReadWriteRParam
// To Start read or write, set inpult values and call action read/write. Busy and Done show the status of the operation
FUNCTION_BLOCK NCiReadWriteRParam EXTENDS FbBase
VAR_OUTPUT CONSTANT
	FNC_READ												:	INT := 0;
	FNC_WRITE												:	INT := 1;
END_VAR         											
VAR_INPUT       											
	Fnc														:	INT (FNC_READ..FNC_WRITE) := FNC_READ;
  	pAddr    												: 	PVOID; //Address of parameter destination variable
   	Index   												: 	DINT; //Index to parameter to read
   	Count   												: 	DINT; //
	rNCIRef													:	REFERENCE TO NCI_REF := 0;
END_VAR
VAR_OUTPUT
END_VAR
VAR
(* cache *******************************************************************)
	MemFnc													:	INT := -1;

(* trigger *****************************************************************)

(* function-block instances	************************************************)
	ItpReadRParamsEx										:	ItpReadRParamsEx := (tTimeout := DEFAULT_ADS_TIMEOUT);
	ItpWriteRParamsEx										:	ItpWriteRParamsEx := (tTimeout := DEFAULT_ADS_TIMEOUT);

END_VAR

	(* Read/Write Nci group R parameter													*)
	(************************************************************************************)

(* Execute ******************************************************************************)
	rtExecute(CLK := Execute);
	IF rtExecute.Q
		AND MemFnc < 0
	THEN
		MemFnc 												:= SEL(Fnc = FNC_WRITE, FNC_READ , FNC_WRITE) ;
		Busy												:= TRUE;
		Done												:= FALSE;
		Error												:= FALSE;
		ErrorID												:= 0;
	END_IF

